LIN {X 0,Y 523.335,Z 480.946,A -85,B 0,C 180,E1 -4767.691,E2 -4767.691} C_VEL
LIN {X 0,Y 523.25,Z 482.542,A -85,B 0,C 180,E1 -4769.231,E2 -4769.231} C_VEL
LIN {X 0,Y 523.247,Z 482.758,A -85,B 0,C 180,E1 -4770,E2 -4770} C_VEL
LIN {X 0,Y 523.275,Z 481.937,A -85,B 0,C 180,E1 -4771.539,E2 -4771.539} C_VEL
LIN {X 0,Y 523.335,Z 480.945,A -85,B 0,C 180,E1 -4772.309,E2 -4772.309} C_VEL
LIN {X 0,Y 523.369,Z 479.554,A -85,B 0,C 180,E1 -4773.079,E2 -4773.079} C_VEL
LIN {X 0,Y 523.425,Z 476.628,A -85,B 0,C 180,E1 -4774.235,E2 -4774.235} C_VEL
LIN {X 0,Y 523.462,Z 472.665,A -85,B 0,C 180,E1 -4775.393,E2 -4775.393} C_VEL
LIN {X 0,Y 523.507,Z 466.591,A -85,B 0,C 180,E1 -4776.742,E2 -4776.742} C_VEL
LIN {X 0,Y 523.676,Z 459.903,A -85,B 0,C 180,E1 -4777.907,E2 -4777.907} C_VEL
LIN {X 0,Y 523.862,Z 451.631,A -85,B 0,C 180,E1 -4779.07,E2 -4779.07} C_VEL
LIN {X 0,Y 524.082,Z 443.149,A -85,B 0,C 180,E1 -4780.04,E2 -4780.04} C_VEL
LIN {X 0,Y 524.37,Z 432.664,A -85,B 0,C 180,E1 -4781.011,E2 -4781.011} C_VEL
LIN {X 0,Y 524.659,Z 422.41,A -85,B 0,C 180,E1 -4781.779,E2 -4781.779} C_VEL
LIN {X 0,Y 524.937,Z 410.907,A -85,B 0,C 180,E1 -4782.468,E2 -4782.468} C_VEL
LIN {X 0,Y 525.162,Z 399.206,A -85,B 0,C 180,E1 -4783.003,E2 -4783.003} C_VEL
LIN {X 0,Y 525.398,Z 385.719,A -85,B 0,C 180,E1 -4783.44,E2 -4783.44} C_VEL
LIN {X 0,Y 525.556,Z 372.288,A -85,B 0,C 180,E1 -4783.706,E2 -4783.706} C_VEL
LIN {X 0,Y 525.863,Z 280.733,A -85,B 0,C 180,E1 -4784.966,E2 -4784.966} C_VEL
LIN {X 0,Y 524.292,Z 270.902,A -85,B 0,C 180,E1 -4785.169,E2 -4785.169} C_VEL
LIN {X 0,Y 524.363,Z 264.633,A -85,B 0,C 180,E1 -4786.148,E2 -4786.148} C_VEL
LIN {X 0,Y 524.69,Z 248.812,A -85,B 0,C 180,E1 -4788.752,E2 -4788.752} C_VEL
LIN {X 0,Y 525.199,Z 230.548,A -85,B 0,C 180,E1 -4791.798,E2 -4791.798} C_VEL
LIN {X 0,Y 524.728,Z 225.858,A -85,B 0,C 180,E1 -4792.616,E2 -4792.616} C_VEL
LIN {X 0,Y 523.966,Z 221.81,A -85,B 0,C 180,E1 -4793.387,E2 -4793.387} C_VEL
LIN {X 0,Y 523.946,Z 221.721,A -85,B 0,C 180,E1 -4796.273,E2 -4796.273} C_VEL
LIN {X 0,Y 523.937,Z 221.717,A -85,B 0,C 180,E1 -4798.875,E2 -4798.875} C_VEL
LIN {X 0,Y 523.927,Z 221.72,A -85,B 0,C 180,E1 -4801.544,E2 -4801.544} C_VEL
LIN {X 0,Y 523.939,Z 221.722,A -85,B 0,C 180,E1 -4804.29,E2 -4804.29} C_VEL
LIN {X 0,Y 523.913,Z 221.719,A -85,B 0,C 180,E1 -4807.132,E2 -4807.132} C_VEL
LIN {X 0,Y 523.923,Z 221.723,A -85,B 0,C 180,E1 -4810.126,E2 -4810.126} C_VEL
LIN {X 0,Y 523.926,Z 221.721,A -85,B 0,C 180,E1 -4812.456,E2 -4812.456} C_VEL
LIN {X 0,Y 523.947,Z 221.715,A -85,B 0,C 180,E1 -4815.31,E2 -4815.31} C_VEL
LIN {X 0,Y 523.95,Z 221.721,A -85,B 0,C 180,E1 -4818.691,E2 -4818.691} C_VEL
LIN {X 0,Y 523.922,Z 221.717,A -85,B 0,C 180,E1 -4821.896,E2 -4821.896} C_VEL
LIN {X 0,Y 523.927,Z 221.725,A -85,B 0,C 180,E1 -4824.911,E2 -4824.911} C_VEL
LIN {X 0,Y 523.943,Z 221.713,A -85,B 0,C 180,E1 -4827.678,E2 -4827.678} C_VEL
LIN {X 0,Y 523.945,Z 221.72,A -85,B 0,C 180,E1 -4830.678,E2 -4830.678} C_VEL
LIN {X 0,Y 523.912,Z 221.72,A -85,B 0,C 180,E1 -4833.723,E2 -4833.723} C_VEL
LIN {X 0,Y 523.916,Z 221.716,A -85,B 0,C 180,E1 -4836.267,E2 -4836.267} C_VEL
LIN {X 0,Y 523.951,Z 221.716,A -85,B 0,C 180,E1 -4838.764,E2 -4838.764} C_VEL
LIN {X 0,Y 523.953,Z 221.718,A -85,B 0,C 180,E1 -4841.218,E2 -4841.218} C_VEL
LIN {X 0,Y 523.934,Z 221.72,A -85,B 0,C 180,E1 -4843.636,E2 -4843.636} C_VEL
LIN {X 0,Y 523.935,Z 221.719,A -85,B 0,C 180,E1 -4846.025,E2 -4846.025} C_VEL
LIN {X 0,Y 523.997,Z 221.709,A -85,B 0,C 180,E1 -4849.174,E2 -4849.174} C_VEL
LIN {X 0,Y 524.002,Z 221.709,A -85,B 0,C 180,E1 -4852.289,E2 -4852.289} C_VEL
LIN {X 0,Y 524.071,Z 221.698,A -85,B 0,C 180,E1 -4854.61,E2 -4854.61} C_VEL
LIN {X 0,Y 524.11,Z 221.699,A -85,B 0,C 180,E1 -4857.691,E2 -4857.691} C_VEL
LIN {X 0,Y 524.116,Z 221.694,A -85,B 0,C 180,E1 -4860.765,E2 -4860.765} C_VEL
LIN {X 0,Y 524.037,Z 221.7,A -85,B 0,C 180,E1 -4863.072,E2 -4863.072} C_VEL
LIN {X 0,Y 524.025,Z 221.713,A -85,B 0,C 180,E1 -4866.156,E2 -4866.156} C_VEL
LIN {X 0,Y 523.982,Z 221.71,A -85,B 0,C 180,E1 -4869.258,E2 -4869.258} C_VEL
LIN {X 0,Y 523.993,Z 221.706,A -85,B 0,C 180,E1 -4871.734,E2 -4871.734} C_VEL
LIN {X 0,Y 523.985,Z 221.711,A -85,B 0,C 180,E1 -4875.049,E2 -4875.049} C_VEL
LIN {X 0,Y 523.936,Z 221.716,A -85,B 0,C 180,E1 -4877.965,E2 -4877.965} C_VEL
LIN {X 0,Y 523.96,Z 221.717,A -85,B 0,C 180,E1 -4880.406,E2 -4880.406} C_VEL
LIN {X 0,Y 523.905,Z 221.728,A -85,B 0,C 180,E1 -4882.889,E2 -4882.889} C_VEL
LIN {X 0,Y 523.935,Z 221.713,A -85,B 0,C 180,E1 -4885.414,E2 -4885.414} C_VEL
LIN {X 0,Y 523.951,Z 221.714,A -85,B 0,C 180,E1 -4887.995,E2 -4887.995} C_VEL
LIN {X 0,Y 523.923,Z 221.721,A -85,B 0,C 180,E1 -4890.851,E2 -4890.851} C_VEL
LIN {X 0,Y 523.938,Z 221.718,A -85,B 0,C 180,E1 -4893.731,E2 -4893.731} C_VEL
LIN {X 0,Y 523.896,Z 221.721,A -85,B 0,C 180,E1 -4896.4,E2 -4896.4} C_VEL
LIN {X 0,Y 523.934,Z 221.719,A -85,B 0,C 180,E1 -4899.077,E2 -4899.077} C_VEL
LIN {X 0,Y 523.935,Z 221.719,A -85,B 0,C 180,E1 -4902.114,E2 -4902.114} C_VEL
LIN {X 0,Y 523.922,Z 221.723,A -85,B 0,C 180,E1 -4905.305,E2 -4905.305} C_VEL
LIN {X 0,Y 523.889,Z 221.724,A -85,B 0,C 180,E1 -4906.894,E2 -4906.894} C_VEL
LIN {X 0,Y 523.214,Z 221.816,A -85,B 0,C 180,E1 -4907.536,E2 -4907.536} C_VEL
LIN {X 0,Y 520.346,Z 222.167,A -85,B 0,C 180,E1 -4908.578,E2 -4908.578} C_VEL
LIN {X 0,Y 517.961,Z 222.468,A -85,B 0,C 180,E1 -4909.417,E2 -4909.417} C_VEL
LIN {X 0,Y 516.989,Z 222.591,A -85,B 0,C 180,E1 -4910.065,E2 -4910.065} C_VEL
LIN {X 0,Y 516.937,Z 222.597,A -85,B 0,C 180,E1 -4910.284,E2 -4910.284} C_VEL
LIN {X 0,Y 516.957,Z 222.758,A -85,B 0,C 180,E1 -4910.489,E2 -4910.489} C_VEL
LIN {X 0,Y 517.786,Z 229.073,A -85,B 0,C 180,E1 -4911.688,E2 -4911.688} C_VEL
LIN {X 0,Y 517.418,Z 247.056,A -85,B 0,C 180,E1 -4914.887,E2 -4914.887} C_VEL
LIN {X 0,Y 517.241,Z 257.287,A -85,B 0,C 180,E1 -4916.658,E2 -4916.658} C_VEL
LIN {X 0,Y 518.403,Z 263.881,A -85,B 0,C 180,E1 -4916.818,E2 -4916.818} C_VEL
LIN {X 0,Y 519.11,Z 269.37,A -85,B 0,C 180,E1 -4916.917,E2 -4916.917} C_VEL
LIN {X 0,Y 518.609,Z 364.635,A -85,B 0,C 180,E1 -4918.261,E2 -4918.261} C_VEL
LIN {X 0,Y 518.423,Z 378.207,A -85,B 0,C 180,E1 -4918.618,E2 -4918.618} C_VEL
LIN {X 0,Y 518.169,Z 390.312,A -85,B 0,C 180,E1 -4919.089,E2 -4919.089} C_VEL
LIN {X 0,Y 517.891,Z 402.731,A -85,B 0,C 180,E1 -4919.748,E2 -4919.748} C_VEL
LIN {X 0,Y 517.6,Z 413.253,A -85,B 0,C 180,E1 -4920.465,E2 -4920.465} C_VEL
LIN {X 0,Y 517.267,Z 424.093,A -85,B 0,C 180,E1 -4921.384,E2 -4921.384} C_VEL
LIN {X 0,Y 517.051,Z 432.491,A -85,B 0,C 180,E1 -4922.259,E2 -4922.259} C_VEL
LIN {X 0,Y 516.749,Z 440.994,A -85,B 0,C 180,E1 -4923.332,E2 -4923.332} C_VEL
LIN {X 0,Y 516.558,Z 449.157,A -85,B 0,C 180,E1 -4924.623,E2 -4924.623} C_VEL
LIN {X 0,Y 516.41,Z 455.564,A -85,B 0,C 180,E1 -4925.903,E2 -4925.903} C_VEL
LIN {X 0,Y 516.327,Z 460.463,A -85,B 0,C 180,E1 -4927.174,E2 -4927.174} C_VEL
LIN {X 0,Y 516.259,Z 464.071,A -85,B 0,C 180,E1 -4928.435,E2 -4928.435} C_VEL
LIN {X 0,Y 516.237,Z 466.879,A -85,B 0,C 180,E1 -4929.927,E2 -4929.927} C_VEL
LIN {X 0,Y 516.172,Z 467.939,A -85,B 0,C 180,E1 -4930.927,E2 -4930.927} C_VEL
LIN {X 0,Y 516.18,Z 468.302,A -85,B 0,C 180,E1 -4932.359,E2 -4932.359} C_VEL
LIN {X 0,Y 516.19,Z 467.766,A -85,B 0,C 180,E1 -4933.386,E2 -4933.386} C_VEL
LIN {X 0,Y 516.209,Z 466.822,A -85,B 0,C 180,E1 -4934.199,E2 -4934.199} C_VEL
LIN {X 0,Y 516.252,Z 465.267,A -85,B 0,C 180,E1 -4935.117,E2 -4935.117} C_VEL
LIN {X 0,Y 516.304,Z 462.587,A -85,B 0,C 180,E1 -4936.219,E2 -4936.219} C_VEL
LIN {X 0,Y 516.341,Z 458.654,A -85,B 0,C 180,E1 -4937.421,E2 -4937.421} C_VEL
LIN {X 0,Y 516.533,Z 453.072,A -85,B 0,C 180,E1 -4938.722,E2 -4938.722} C_VEL
LIN {X 0,Y 516.64,Z 445.925,A -85,B 0,C 180,E1 -4940.012,E2 -4940.012} C_VEL
LIN {X 0,Y 516.839,Z 437.679,A -85,B 0,C 180,E1 -4941.2,E2 -4941.2} C_VEL
LIN {X 0,Y 517.127,Z 429.239,A -85,B 0,C 180,E1 -4942.189,E2 -4942.189} C_VEL
LIN {X 0,Y 517.396,Z 418.866,A -85,B 0,C 180,E1 -4943.174,E2 -4943.174} C_VEL
LIN {X 0,Y 517.748,Z 407.176,A -85,B 0,C 180,E1 -4944.059,E2 -4944.059} C_VEL
LIN {X 0,Y 518.06,Z 395.541,A -85,B 0,C 180,E1 -4944.746,E2 -4944.746} C_VEL
LIN {X 0,Y 518.319,Z 383.483,A -85,B 0,C 180,E1 -4945.285,E2 -4945.285} C_VEL
LIN {X 0,Y 518.506,Z 370.393,A -85,B 0,C 180,E1 -4945.7,E2 -4945.7} C_VEL
LIN {X 0,Y 518.683,Z 357.572,A -85,B 0,C 180,E1 -4945.945,E2 -4945.945} C_VEL
LIN {X 0,Y 519.048,Z 267.685,A -85,B 0,C 180,E1 -4947.199,E2 -4947.199} C_VEL
LIN {X 0,Y 517.307,Z 257.515,A -85,B 0,C 180,E1 -4947.42,E2 -4947.42} C_VEL
LIN {X 0,Y 517.358,Z 249.489,A -85,B 0,C 180,E1 -4948.832,E2 -4948.832} C_VEL
LIN {X 0,Y 517.835,Z 233.569,A -85,B 0,C 180,E1 -4951.75,E2 -4951.75} C_VEL
LIN {X 0,Y 517.797,Z 227.316,A -85,B 0,C 180,E1 -4952.917,E2 -4952.917} C_VEL
LIN {X 0,Y 516.879,Z 222.661,A -85,B 0,C 180,E1 -4953.874,E2 -4953.874} C_VEL
LIN {X 0,Y 517.008,Z 222.587,A -85,B 0,C 180,E1 -4956.243,E2 -4956.243} C_VEL
LIN {X 0,Y 516.947,Z 222.595,A -85,B 0,C 180,E1 -4958.6,E2 -4958.6} C_VEL
LIN {X 0,Y 516.967,Z 222.585,A -85,B 0,C 180,E1 -4961.844,E2 -4961.844} C_VEL
LIN {X 0,Y 516.928,Z 222.592,A -85,B 0,C 180,E1 -4965.162,E2 -4965.162} C_VEL
LIN {X 0,Y 516.883,Z 222.594,A -85,B 0,C 180,E1 -4968.223,E2 -4968.223} C_VEL
LIN {X 0,Y 516.888,Z 222.595,A -85,B 0,C 180,E1 -4970.702,E2 -4970.702} C_VEL
LIN {X 0,Y 516.873,Z 222.601,A -85,B 0,C 180,E1 -4973.223,E2 -4973.223} C_VEL
LIN {X 0,Y 516.909,Z 222.582,A -85,B 0,C 180,E1 -4976.202,E2 -4976.202} C_VEL
LIN {X 0,Y 516.9,Z 222.596,A -85,B 0,C 180,E1 -4979.305,E2 -4979.305} C_VEL
LIN {X 0,Y 516.86,Z 222.599,A -85,B 0,C 180,E1 -4982.025,E2 -4982.025} C_VEL
LIN {X 0,Y 516.894,Z 222.591,A -85,B 0,C 180,E1 -4984.823,E2 -4984.823} C_VEL
LIN {X 0,Y 516.857,Z 222.602,A -85,B 0,C 180,E1 -4987.949,E2 -4987.949} C_VEL
LIN {X 0,Y 516.885,Z 222.592,A -85,B 0,C 180,E1 -4990.741,E2 -4990.741} C_VEL
LIN {X 0,Y 516.918,Z 222.596,A -85,B 0,C 180,E1 -4993.905,E2 -4993.905} C_VEL
LIN {X 0,Y 516.92,Z 222.597,A -85,B 0,C 180,E1 -4996.108,E2 -4996.108} C_VEL
LIN {X 0,Y 516.884,Z 222.592,A -85,B 0,C 180,E1 -4999.265,E2 -4999.265} C_VEL
LIN {X 0,Y 516.858,Z 222.596,A -85,B 0,C 180,E1 -5002.059,E2 -5002.059} C_VEL
LIN {X 0,Y 516.876,Z 222.594,A -85,B 0,C 180,E1 -5005.181,E2 -5005.181} C_VEL
LIN {X 0,Y 516.859,Z 222.6,A -85,B 0,C 180,E1 -5007.98,E2 -5007.98} C_VEL
LIN {X 0,Y 516.913,Z 222.588,A -85,B 0,C 180,E1 -5010.7,E2 -5010.7} C_VEL
LIN {X 0,Y 516.924,Z 222.582,A -85,B 0,C 180,E1 -5013.807,E2 -5013.807} C_VEL
LIN {X 0,Y 516.874,Z 222.604,A -85,B 0,C 180,E1 -5016.782,E2 -5016.782} C_VEL
LIN {X 0,Y 516.923,Z 222.588,A -85,B 0,C 180,E1 -5019.735,E2 -5019.735} C_VEL
LIN {X 0,Y 516.917,Z 222.589,A -85,B 0,C 180,E1 -5022.6,E2 -5022.6} C_VEL
LIN {X 0,Y 516.929,Z 222.585,A -85,B 0,C 180,E1 -5025.034,E2 -5025.034} C_VEL
LIN {X 0,Y 516.994,Z 222.577,A -85,B 0,C 180,E1 -5028.238,E2 -5028.238} C_VEL
LIN {X 0,Y 516.965,Z 222.592,A -85,B 0,C 180,E1 -5031.404,E2 -5031.404} C_VEL
LIN {X 0,Y 517.008,Z 222.58,A -85,B 0,C 180,E1 -5033.761,E2 -5033.761} C_VEL
LIN {X 0,Y 517.079,Z 222.566,A -85,B 0,C 180,E1 -5037.667,E2 -5037.667} C_VEL
LIN {X 0,Y 517.09,Z 222.564,A -85,B 0,C 180,E1 -5040.782,E2 -5040.782} C_VEL
LIN {X 0,Y 517.01,Z 222.578,A -85,B 0,C 180,E1 -5043.12,E2 -5043.12} C_VEL
LIN {X 0,Y 516.992,Z 222.583,A -85,B 0,C 180,E1 -5046.247,E2 -5046.247} C_VEL
LIN {X 0,Y 516.965,Z 222.578,A -85,B 0,C 180,E1 -5048.604,E2 -5048.604} C_VEL
LIN {X 0,Y 516.954,Z 222.582,A -85,B 0,C 180,E1 -5051.81,E2 -5051.81} C_VEL
LIN {X 0,Y 516.948,Z 222.586,A -85,B 0,C 180,E1 -5055.149,E2 -5055.149} C_VEL
LIN {X 0,Y 516.92,Z 222.596,A -85,B 0,C 180,E1 -5058.225,E2 -5058.225} C_VEL
LIN {X 0,Y 516.917,Z 222.59,A -85,B 0,C 180,E1 -5060.704,E2 -5060.704} C_VEL
LIN {X 0,Y 516.906,Z 222.592,A -85,B 0,C 180,E1 -5064.075,E2 -5064.075} C_VEL
LIN {X 0,Y 516.909,Z 222.6,A -85,B 0,C 180,E1 -5066.661,E2 -5066.661} C_VEL
LIN {X 0,Y 516.915,Z 222.585,A -85,B 0,C 180,E1 -5069.525,E2 -5069.525} C_VEL
LIN {X 0,Y 516.9,Z 222.595,A -85,B 0,C 180,E1 -5072.545,E2 -5072.545} C_VEL
LIN {X 0,Y 516.869,Z 222.6,A -85,B 0,C 180,E1 -5075.331,E2 -5075.331} C_VEL
LIN {X 0,Y 516.884,Z 222.592,A -85,B 0,C 180,E1 -5077.944,E2 -5077.944} C_VEL
LIN {X 0,Y 516.889,Z 222.596,A -85,B 0,C 180,E1 -5080.743,E2 -5080.743} C_VEL
LIN {X 0,Y 516.888,Z 222.586,A -85,B 0,C 180,E1 -5083.905,E2 -5083.905} C_VEL
LIN {X 0,Y 516.887,Z 222.589,A -85,B 0,C 180,E1 -5086.109,E2 -5086.109} C_VEL
LIN {X 0,Y 516.889,Z 222.597,A -85,B 0,C 180,E1 -5089.259,E2 -5089.259} C_VEL
LIN {X 0,Y 516.867,Z 222.597,A -85,B 0,C 180,E1 -5092.275,E2 -5092.275} C_VEL
LIN {X 0,Y 516.888,Z 222.595,A -85,B 0,C 180,E1 -5095.176,E2 -5095.176} C_VEL
LIN {X 0,Y 516.88,Z 222.603,A -85,B 0,C 180,E1 -5097.976,E2 -5097.976} C_VEL
LIN {X 0,Y 516.926,Z 222.592,A -85,B 0,C 180,E1 -5100.696,E2 -5100.696} C_VEL
LIN {X 0,Y 516.913,Z 222.594,A -85,B 0,C 180,E1 -5103.342,E2 -5103.342} C_VEL
LIN {X 0,Y 516.939,Z 222.71,A -85,B 0,C 180,E1 -5106.409,E2 -5106.409} C_VEL
LIN {X 0,Y 518.257,Z 230.708,A -85,B 0,C 180,E1 -5107.895,E2 -5107.895} C_VEL
LIN {X 0,Y 517.79,Z 248.894,A -85,B 0,C 180,E1 -5110.989,E2 -5110.989} C_VEL
LIN {X 0,Y 517.375,Z 265.834,A -85,B 0,C 180,E1 -5113.831,E2 -5113.831} C_VEL
LIN {X 0,Y 517.277,Z 270.785,A -85,B 0,C 180,E1 -5114.615,E2 -5114.615} C_VEL
LIN {X 0,Y 518.992,Z 281.529,A -85,B 0,C 180,E1 -5114.844,E2 -5114.844} C_VEL
LIN {X 0,Y 518.631,Z 378.172,A -85,B 0,C 180,E1 -5116.207,E2 -5116.207} C_VEL
LIN {X 0,Y 518.407,Z 391.541,A -85,B 0,C 180,E1 -5116.551,E2 -5116.551} C_VEL
LIN {X 0,Y 518.138,Z 404.876,A -85,B 0,C 180,E1 -5117.068,E2 -5117.068} C_VEL
LIN {X 0,Y 517.878,Z 416.116,A -85,B 0,C 180,E1 -5117.662,E2 -5117.662} C_VEL
LIN {X 0,Y 517.568,Z 427.664,A -85,B 0,C 180,E1 -5118.446,E2 -5118.446} C_VEL
LIN {X 0,Y 517.205,Z 438.107,A -85,B 0,C 180,E1 -5119.331,E2 -5119.331} C_VEL
LIN {X 0,Y 516.98,Z 446.645,A -85,B 0,C 180,E1 -5120.217,E2 -5120.217} C_VEL
LIN {X 0,Y 516.755,Z 454.519,A -85,B 0,C 180,E1 -5121.199,E2 -5121.199} C_VEL
LIN {X 0,Y 516.552,Z 462.207,A -85,B 0,C 180,E1 -5122.377,E2 -5122.377} C_VEL
LIN {X 0,Y 516.405,Z 469.291,A -85,B 0,C 180,E1 -5123.75,E2 -5123.75} C_VEL
LIN {X 0,Y 516.314,Z 474.002,A -85,B 0,C 180,E1 -5124.924,E2 -5124.924} C_VEL
LIN {X 0,Y 516.353,Z 477.601,A -85,B 0,C 180,E1 -5126.098,E2 -5126.098} C_VEL
LIN {X 0,Y 516.284,Z 479.456,A -85,B 0,C 180,E1 -5126.879,E2 -5126.879} C_VEL
LIN {X 0,Y 516.262,Z 480.847,A -85,B 0,C 180,E1 -5127.66,E2 -5127.66} C_VEL
LIN {X 0,Y 516.161,Z 482.444,A -85,B 0,C 180,E1 -5129.22,E2 -5129.22} C_VEL
LIN {X 0,Y 516.155,Z 482.66,A -85,B 0,C 180,E1 -5130,E2 -5130} C_VEL
LIN {X 0,Y 516.193,Z 481.838,A -85,B 0,C 180,E1 -5131.561,E2 -5131.561} C_VEL
LIN {X 0,Y 516.262,Z 480.846,A -85,B 0,C 180,E1 -5132.341,E2 -5132.341} C_VEL
LIN {X 0,Y 516.284,Z 479.454,A -85,B 0,C 180,E1 -5133.122,E2 -5133.122} C_VEL
LIN {X 0,Y 516.314,Z 476.526,A -85,B 0,C 180,E1 -5134.294,E2 -5134.294} C_VEL
LIN {X 0,Y 516.399,Z 472.562,A -85,B 0,C 180,E1 -5135.467,E2 -5135.467} C_VEL
LIN {X 0,Y 516.426,Z 467.354,A -85,B 0,C 180,E1 -5136.665,E2 -5136.665} C_VEL
LIN {X 0,Y 516.585,Z 461.031,A -85,B 0,C 180,E1 -5137.819,E2 -5137.819} C_VEL
LIN {X 0,Y 516.773,Z 453.011,A -85,B 0,C 180,E1 -5138.998,E2 -5138.998} C_VEL
LIN {X 0,Y 517.027,Z 444.837,A -85,B 0,C 180,E1 -5139.981,E2 -5139.981} C_VEL
LIN {X 0,Y 517.337,Z 434.865,A -85,B 0,C 180,E1 -5140.964,E2 -5140.964} C_VEL
LIN {X 0,Y 517.649,Z 425.021,A -85,B 0,C 180,E1 -5141.751,E2 -5141.751} C_VEL
LIN {X 0,Y 517.917,Z 413.872,A -85,B 0,C 180,E1 -5142.466,E2 -5142.466} C_VEL
LIN {X 0,Y 518.192,Z 401.434,A -85,B 0,C 180,E1 -5143.081,E2 -5143.081} C_VEL
LIN {X 0,Y 518.487,Z 388.315,A -85,B 0,C 180,E1 -5143.547,E2 -5143.547} C_VEL
LIN {X 0,Y 518.654,Z 375.175,A -85,B 0,C 180,E1 -5143.842,E2 -5143.842} C_VEL
LIN {X 0,Y 518.988,Z 281.442,A -85,B 0,C 180,E1 -5145.157,E2 -5145.157} C_VEL
LIN {X 0,Y 517.261,Z 270.8,A -85,B 0,C 180,E1 -5145.38,E2 -5145.38} C_VEL
LIN {X 0,Y 517.493,Z 259.66,A -85,B 0,C 180,E1 -5147.181,E2 -5147.181} C_VEL
LIN {X 0,Y 517.948,Z 241.633,A -85,B 0,C 180,E1 -5150.206,E2 -5150.206} C_VEL
LIN {X 0,Y 518.247,Z 230.459,A -85,B 0,C 180,E1 -5152.106,E2 -5152.106} C_VEL
LIN {X 0,Y 516.934,Z 222.727,A -85,B 0,C 180,E1 -5153.539,E2 -5153.539} C_VEL
LIN {X 0,Y 516.914,Z 222.594,A -85,B 0,C 180,E1 -5156.659,E2 -5156.659} C_VEL
LIN {X 0,Y 516.916,Z 222.595,A -85,B 0,C 180,E1 -5159.522,E2 -5159.522} C_VEL
LIN {X 0,Y 516.905,Z 222.593,A -85,B 0,C 180,E1 -5162.542,E2 -5162.542} C_VEL
LIN {X 0,Y 516.871,Z 222.596,A -85,B 0,C 180,E1 -5165.328,E2 -5165.328} C_VEL
LIN {X 0,Y 516.887,Z 222.601,A -85,B 0,C 180,E1 -5167.942,E2 -5167.942} C_VEL
LIN {X 0,Y 516.874,Z 222.599,A -85,B 0,C 180,E1 -5170.743,E2 -5170.743} C_VEL
LIN {X 0,Y 516.864,Z 222.598,A -85,B 0,C 180,E1 -5172.833,E2 -5172.833} C_VEL
LIN {X 0,Y 516.906,Z 222.594,A -85,B 0,C 180,E1 -5175.006,E2 -5175.006} C_VEL
LIN {X 0,Y 516.913,Z 222.592,A -85,B 0,C 180,E1 -5178.399,E2 -5178.399} C_VEL
LIN {X 0,Y 516.888,Z 222.594,A -85,B 0,C 180,E1 -5181.282,E2 -5181.282} C_VEL
LIN {X 0,Y 516.875,Z 222.597,A -85,B 0,C 180,E1 -5184.218,E2 -5184.218} C_VEL
LIN {X 0,Y 516.89,Z 222.599,A -85,B 0,C 180,E1 -5187.05,E2 -5187.05} C_VEL
LIN {X 0,Y 516.876,Z 222.596,A -85,B 0,C 180,E1 -5189.793,E2 -5189.793} C_VEL
LIN {X 0,Y 516.884,Z 222.594,A -85,B 0,C 180,E1 -5192.462,E2 -5192.462} C_VEL
LIN {X 0,Y 516.854,Z 222.606,A -85,B 0,C 180,E1 -5195.066,E2 -5195.066} C_VEL
LIN {X 0,Y 516.878,Z 222.599,A -85,B 0,C 180,E1 -5197.619,E2 -5197.619} C_VEL
LIN {X 0,Y 516.939,Z 222.585,A -85,B 0,C 180,E1 -5200.127,E2 -5200.127} C_VEL
LIN {X 0,Y 516.913,Z 222.591,A -85,B 0,C 180,E1 -5202.593,E2 -5202.593} C_VEL
LIN {X 0,Y 516.948,Z 222.585,A -85,B 0,C 180,E1 -5205.027,E2 -5205.027} C_VEL
LIN {X 0,Y 516.972,Z 222.582,A -85,B 0,C 180,E1 -5208.231,E2 -5208.231} C_VEL
LIN {X 0,Y 516.934,Z 222.592,A -85,B 0,C 180,E1 -5211.396,E2 -5211.396} C_VEL
LIN {X 0,Y 516.989,Z 222.587,A -85,B 0,C 180,E1 -5213.753,E2 -5213.753} C_VEL
LIN {X 0,Y 516.975,Z 222.582,A -85,B 0,C 180,E1 -5216.879,E2 -5216.879} C_VEL
LIN {X 0,Y 517.091,Z 222.566,A -85,B 0,C 180,E1 -5219.218,E2 -5219.218} C_VEL
LIN {X 0,Y 517.079,Z 222.573,A -85,B 0,C 180,E1 -5222.333,E2 -5222.333} C_VEL
LIN {X 0,Y 517.018,Z 222.578,A -85,B 0,C 180,E1 -5225.456,E2 -5225.456} C_VEL
LIN {X 0,Y 516.959,Z 222.591,A -85,B 0,C 180,E1 -5228.597,E2 -5228.597} C_VEL
LIN {X 0,Y 516.945,Z 222.585,A -85,B 0,C 180,E1 -5231.803,E2 -5231.803} C_VEL
LIN {X 0,Y 516.938,Z 222.588,A -85,B 0,C 180,E1 -5235.143,E2 -5235.143} C_VEL
LIN {X 0,Y 516.905,Z 222.594,A -85,B 0,C 180,E1 -5238.218,E2 -5238.218} C_VEL
LIN {X 0,Y 516.901,Z 222.601,A -85,B 0,C 180,E1 -5240.697,E2 -5240.697} C_VEL
LIN {X 0,Y 516.859,Z 222.602,A -85,B 0,C 180,E1 -5243.219,E2 -5243.219} C_VEL
LIN {X 0,Y 516.925,Z 222.584,A -85,B 0,C 180,E1 -5246.192,E2 -5246.192} C_VEL
LIN {X 0,Y 516.901,Z 222.597,A -85,B 0,C 180,E1 -5249.3,E2 -5249.3} C_VEL
LIN {X 0,Y 516.875,Z 222.596,A -85,B 0,C 180,E1 -5252.54,E2 -5252.54} C_VEL
LIN {X 0,Y 516.857,Z 222.603,A -85,B 0,C 180,E1 -5255.328,E2 -5255.328} C_VEL
LIN {X 0,Y 516.858,Z 222.598,A -85,B 0,C 180,E1 -5257.94,E2 -5257.94} C_VEL
LIN {X 0,Y 516.888,Z 222.595,A -85,B 0,C 180,E1 -5260.734,E2 -5260.734} C_VEL
LIN {X 0,Y 516.85,Z 222.605,A -85,B 0,C 180,E1 -5263.899,E2 -5263.899} C_VEL
LIN {X 0,Y 516.848,Z 222.604,A -85,B 0,C 180,E1 -5266.103,E2 -5266.103} C_VEL
LIN {X 0,Y 516.884,Z 222.6,A -85,B 0,C 180,E1 -5269.258,E2 -5269.258} C_VEL
LIN {X 0,Y 516.937,Z 222.597,A -85,B 0,C 180,E1 -5270.284,E2 -5270.284} C_VEL
LIN {X 0,Y 516.819,Z 223.447,A -85,B 0,C 180,E1 -5270.614,E2 -5270.614} C_VEL
LIN {X 0,Y 516.039,Z 226.233,A -85,B 0,C 180,E1 -5271.103,E2 -5271.103} C_VEL
LIN {X 0,Y 511.302,Z 236.065,A -85,B 0,C 180,E1 -5272.666,E2 -5272.666} C_VEL
LIN {X 0,Y 510.587,Z 239.154,A -85,B 0,C 180,E1 -5273.217,E2 -5273.217} C_VEL
LIN {X 0,Y 510.32,Z 254.146,A -85,B 0,C 180,E1 -5275.906,E2 -5275.906} C_VEL
LIN {X 0,Y 510.255,Z 257.328,A -85,B 0,C 180,E1 -5276.435,E2 -5276.435} C_VEL
LIN {X 0,Y 511.252,Z 263.108,A -85,B 0,C 180,E1 -5276.587,E2 -5276.587} C_VEL
LIN {X 0,Y 512.281,Z 269.989,A -85,B 0,C 180,E1 -5276.718,E2 -5276.718} C_VEL
LIN {X 0,Y 511.718,Z 365.353,A -85,B 0,C 180,E1 -5278.087,E2 -5278.087} C_VEL
LIN {X 0,Y 511.509,Z 379.166,A -85,B 0,C 180,E1 -5278.463,E2 -5278.463} C_VEL
LIN {X 0,Y 511.238,Z 391.625,A -85,B 0,C 180,E1 -5278.968,E2 -5278.968} C_VEL
LIN {X 0,Y 510.927,Z 403.195,A -85,B 0,C 180,E1 -5279.602,E2 -5279.602} C_VEL
LIN {X 0,Y 510.584,Z 414.686,A -85,B 0,C 180,E1 -5280.409,E2 -5280.409} C_VEL
LIN {X 0,Y 510.219,Z 425.514,A -85,B 0,C 180,E1 -5281.366,E2 -5281.366} C_VEL
LIN {X 0,Y 509.99,Z 433.94,A -85,B 0,C 180,E1 -5282.283,E2 -5282.283} C_VEL
LIN {X 0,Y 509.681,Z 441.999,A -85,B 0,C 180,E1 -5283.345,E2 -5283.345} C_VEL
LIN {X 0,Y 509.483,Z 450.166,A -85,B 0,C 180,E1 -5284.683,E2 -5284.683} C_VEL
LIN {X 0,Y 509.334,Z 456.399,A -85,B 0,C 180,E1 -5285.995,E2 -5285.995} C_VEL
LIN {X 0,Y 509.229,Z 461.063,A -85,B 0,C 180,E1 -5287.267,E2 -5287.267} C_VEL
LIN {X 0,Y 509.182,Z 463.515,A -85,B 0,C 180,E1 -5288.12,E2 -5288.12} C_VEL
LIN {X 0,Y 509.143,Z 465.442,A -85,B 0,C 180,E1 -5288.968,E2 -5288.968} C_VEL
LIN {X 0,Y 509.147,Z 466.858,A -85,B 0,C 180,E1 -5289.813,E2 -5289.813} C_VEL
LIN {X 0,Y 509.109,Z 467.834,A -85,B 0,C 180,E1 -5290.652,E2 -5290.652} C_VEL
LIN {X 0,Y 509.072,Z 468.353,A -85,B 0,C 180,E1 -5291.486,E2 -5291.486} C_VEL
LIN {X 0,Y 509.102,Z 468.409,A -85,B 0,C 180,E1 -5292.32,E2 -5292.32} C_VEL
LIN {X 0,Y 509.091,Z 468.053,A -85,B 0,C 180,E1 -5293.148,E2 -5293.148} C_VEL
LIN {X 0,Y 509.096,Z 467.28,A -85,B 0,C 180,E1 -5293.972,E2 -5293.972} C_VEL
LIN {X 0,Y 509.18,Z 465.595,A -85,B 0,C 180,E1 -5295.033,E2 -5295.033} C_VEL
LIN {X 0,Y 509.202,Z 462.271,A -85,B 0,C 180,E1 -5296.43,E2 -5296.43} C_VEL
LIN {X 0,Y 509.288,Z 458.192,A -85,B 0,C 180,E1 -5297.649,E2 -5297.649} C_VEL
LIN {X 0,Y 509.443,Z 451.908,A -85,B 0,C 180,E1 -5299.065,E2 -5299.065} C_VEL
LIN {X 0,Y 509.613,Z 445.083,A -85,B 0,C 180,E1 -5300.274,E2 -5300.274} C_VEL
LIN {X 0,Y 509.924,Z 436.587,A -85,B 0,C 180,E1 -5301.479,E2 -5301.479} C_VEL
LIN {X 0,Y 510.185,Z 426.496,A -85,B 0,C 180,E1 -5302.622,E2 -5302.622} C_VEL
LIN {X 0,Y 510.546,Z 415.986,A -85,B 0,C 180,E1 -5303.578,E2 -5303.578} C_VEL
LIN {X 0,Y 510.881,Z 404.956,A -85,B 0,C 180,E1 -5304.375,E2 -5304.375} C_VEL
LIN {X 0,Y 511.235,Z 392.614,A -85,B 0,C 180,E1 -5305.071,E2 -5305.071} C_VEL
LIN {X 0,Y 511.483,Z 380.921,A -85,B 0,C 180,E1 -5305.567,E2 -5305.567} C_VEL
LIN {X 0,Y 511.675,Z 368.29,A -85,B 0,C 180,E1 -5305.939,E2 -5305.939} C_VEL
LIN {X 0,Y 511.802,Z 350.571,A -85,B 0,C 180,E1 -5306.235,E2 -5306.235} C_VEL
LIN {X 0,Y 512.128,Z 267.888,A -85,B 0,C 180,E1 -5307.407,E2 -5307.407} C_VEL
LIN {X 0,Y 510.317,Z 257.676,A -85,B 0,C 180,E1 -5307.632,E2 -5307.632} C_VEL
LIN {X 0,Y 510.307,Z 254.132,A -85,B 0,C 180,E1 -5308.224,E2 -5308.224} C_VEL
LIN {X 0,Y 510.721,Z 238.142,A -85,B 0,C 180,E1 -5311.182,E2 -5311.182} C_VEL
LIN {X 0,Y 511.007,Z 229.708,A -85,B 0,C 180,E1 -5312.759,E2 -5312.759} C_VEL
LIN {X 0,Y 509.83,Z 223.535,A -85,B 0,C 180,E1 -5314.026,E2 -5314.026} C_VEL
LIN {X 0,Y 509.973,Z 223.464,A -85,B 0,C 180,E1 -5316.329,E2 -5316.329} C_VEL
LIN {X 0,Y 509.919,Z 223.469,A -85,B 0,C 180,E1 -5318.72,E2 -5318.72} C_VEL
LIN {X 0,Y 509.912,Z 223.465,A -85,B 0,C 180,E1 -5321.931,E2 -5321.931} C_VEL
LIN {X 0,Y 509.893,Z 223.467,A -85,B 0,C 180,E1 -5325.264,E2 -5325.264} C_VEL
LIN {X 0,Y 509.862,Z 223.467,A -85,B 0,C 180,E1 -5328.011,E2 -5328.011} C_VEL
LIN {X 0,Y 509.841,Z 223.478,A -85,B 0,C 180,E1 -5331.002,E2 -5331.002} C_VEL
LIN {X 0,Y 509.827,Z 223.474,A -85,B 0,C 180,E1 -5333.563,E2 -5333.563} C_VEL
LIN {X 0,Y 509.877,Z 223.458,A -85,B 0,C 180,E1 -5336.384,E2 -5336.384} C_VEL
LIN {X 0,Y 509.847,Z 223.467,A -85,B 0,C 180,E1 -5338.846,E2 -5338.846} C_VEL
LIN {X 0,Y 509.815,Z 223.482,A -85,B 0,C 180,E1 -5341.59,E2 -5341.59} C_VEL
LIN {X 0,Y 509.841,Z 223.469,A -85,B 0,C 180,E1 -5344.414,E2 -5344.414} C_VEL
LIN {X 0,Y 509.793,Z 223.481,A -85,B 0,C 180,E1 -5347.342,E2 -5347.342} C_VEL
LIN {X 0,Y 509.851,Z 223.469,A -85,B 0,C 180,E1 -5350.38,E2 -5350.38} C_VEL
LIN {X 0,Y 509.857,Z 223.469,A -85,B 0,C 180,E1 -5353.567,E2 -5353.567} C_VEL
LIN {X 0,Y 509.859,Z 223.472,A -85,B 0,C 180,E1 -5356.44,E2 -5356.44} C_VEL
LIN {X 0,Y 509.847,Z 223.471,A -85,B 0,C 180,E1 -5359.626,E2 -5359.626} C_VEL
LIN {X 0,Y 509.796,Z 223.475,A -85,B 0,C 180,E1 -5362.664,E2 -5362.664} C_VEL
LIN {X 0,Y 509.838,Z 223.473,A -85,B 0,C 180,E1 -5365.8,E2 -5365.8} C_VEL
LIN {X 0,Y 509.824,Z 223.475,A -85,B 0,C 180,E1 -5368.723,E2 -5368.723} C_VEL
LIN {X 0,Y 509.863,Z 223.46,A -85,B 0,C 180,E1 -5371.16,E2 -5371.16} C_VEL
LIN {X 0,Y 509.89,Z 223.458,A -85,B 0,C 180,E1 -5373.833,E2 -5373.833} C_VEL
LIN {X 0,Y 509.832,Z 223.475,A -85,B 0,C 180,E1 -5376.442,E2 -5376.442} C_VEL
LIN {X 0,Y 509.901,Z 223.463,A -85,B 0,C 180,E1 -5379.849,E2 -5379.849} C_VEL
LIN {X 0,Y 509.874,Z 223.463,A -85,B 0,C 180,E1 -5383.179,E2 -5383.179} C_VEL
LIN {X 0,Y 509.852,Z 223.463,A -85,B 0,C 180,E1 -5385.638,E2 -5385.638} C_VEL
LIN {X 0,Y 509.916,Z 223.463,A -85,B 0,C 180,E1 -5388.879,E2 -5388.879} C_VEL
LIN {X 0,Y 509.945,Z 223.458,A -85,B 0,C 180,E1 -5392.082,E2 -5392.082} C_VEL
LIN {X 0,Y 509.979,Z 223.45,A -85,B 0,C 180,E1 -5394.468,E2 -5394.468} C_VEL
LIN {X 0,Y 510.05,Z 223.441,A -85,B 0,C 180,E1 -5397.635,E2 -5397.635} C_VEL
LIN {X 0,Y 510.06,Z 223.44,A -85,B 0,C 180,E1 -5400.793,E2 -5400.793} C_VEL
LIN {X 0,Y 509.952,Z 223.458,A -85,B 0,C 180,E1 -5403.164,E2 -5403.164} C_VEL
LIN {X 0,Y 509.939,Z 223.46,A -85,B 0,C 180,E1 -5406.333,E2 -5406.333} C_VEL
LIN {X 0,Y 509.911,Z 223.455,A -85,B 0,C 180,E1 -5408.723,E2 -5408.723} C_VEL
LIN {X 0,Y 509.906,Z 223.461,A -85,B 0,C 180,E1 -5411.935,E2 -5411.935} C_VEL
LIN {X 0,Y 509.897,Z 223.464,A -85,B 0,C 180,E1 -5415.245,E2 -5415.245} C_VEL
LIN {X 0,Y 509.871,Z 223.47,A -85,B 0,C 180,E1 -5417.996,E2 -5417.996} C_VEL
LIN {X 0,Y 509.891,Z 223.466,A -85,B 0,C 180,E1 -5420.404,E2 -5420.404} C_VEL
LIN {X 0,Y 509.833,Z 223.471,A -85,B 0,C 180,E1 -5423.566,E2 -5423.566} C_VEL
LIN {X 0,Y 509.886,Z 223.471,A -85,B 0,C 180,E1 -5426.374,E2 -5426.374} C_VEL
LIN {X 0,Y 509.878,Z 223.47,A -85,B 0,C 180,E1 -5428.847,E2 -5428.847} C_VEL
LIN {X 0,Y 509.824,Z 223.474,A -85,B 0,C 180,E1 -5431.592,E2 -5431.592} C_VEL
LIN {X 0,Y 509.843,Z 223.473,A -85,B 0,C 180,E1 -5434.417,E2 -5434.417} C_VEL
LIN {X 0,Y 509.814,Z 223.48,A -85,B 0,C 180,E1 -5437.343,E2 -5437.343} C_VEL
LIN {X 0,Y 509.845,Z 223.471,A -85,B 0,C 180,E1 -5440.384,E2 -5440.384} C_VEL
LIN {X 0,Y 509.812,Z 223.477,A -85,B 0,C 180,E1 -5443.061,E2 -5443.061} C_VEL
LIN {X 0,Y 509.829,Z 223.471,A -85,B 0,C 180,E1 -5445.795,E2 -5445.795} C_VEL
LIN {X 0,Y 509.859,Z 223.469,A -85,B 0,C 180,E1 -5448.575,E2 -5448.575} C_VEL
LIN {X 0,Y 509.856,Z 223.474,A -85,B 0,C 180,E1 -5451.788,E2 -5451.788} C_VEL
LIN {X 0,Y 509.834,Z 223.473,A -85,B 0,C 180,E1 -5454.623,E2 -5454.623} C_VEL
LIN {X 0,Y 509.868,Z 223.472,A -85,B 0,C 180,E1 -5457.482,E2 -5457.482} C_VEL
LIN {X 0,Y 509.865,Z 223.475,A -85,B 0,C 180,E1 -5460.275,E2 -5460.275} C_VEL
LIN {X 0,Y 509.88,Z 223.47,A -85,B 0,C 180,E1 -5462.945,E2 -5462.945} C_VEL
LIN {X 0,Y 509.868,Z 223.558,A -85,B 0,C 180,E1 -5466.223,E2 -5466.223} C_VEL
LIN {X 0,Y 511.163,Z 230.597,A -85,B 0,C 180,E1 -5467.572,E2 -5467.572} C_VEL
LIN {X 0,Y 511.1,Z 239.088,A -85,B 0,C 180,E1 -5469.052,E2 -5469.052} C_VEL
LIN {X 0,Y 510.663,Z 256.558,A -85,B 0,C 180,E1 -5472.047,E2 -5472.047} C_VEL
LIN {X 0,Y 510.28,Z 270.687,A -85,B 0,C 180,E1 -5474.398,E2 -5474.398} C_VEL
LIN {X 0,Y 512.223,Z 283.12,A -85,B 0,C 180,E1 -5474.663,E2 -5474.663} C_VEL
LIN {X 0,Y 511.726,Z 379.172,A -85,B 0,C 180,E1 -5476.043,E2 -5476.043} C_VEL
LIN {X 0,Y 511.48,Z 392.931,A -85,B 0,C 180,E1 -5476.416,E2 -5476.416} C_VEL
LIN {X 0,Y 511.175,Z 405.786,A -85,B 0,C 180,E1 -5476.939,E2 -5476.939} C_VEL
LIN {X 0,Y 510.827,Z 418.437,A -85,B 0,C 180,E1 -5477.645,E2 -5477.645} C_VEL
LIN {X 0,Y 510.509,Z 430.112,A -85,B 0,C 180,E1 -5478.486,E2 -5478.486} C_VEL
LIN {X 0,Y 510.152,Z 441.003,A -85,B 0,C 180,E1 -5479.483,E2 -5479.483} C_VEL
LIN {X 0,Y 509.85,Z 449.849,A -85,B 0,C 180,E1 -5480.479,E2 -5480.479} C_VEL
LIN {X 0,Y 509.597,Z 458.475,A -85,B 0,C 180,E1 -5481.674,E2 -5481.674} C_VEL
LIN {X 0,Y 509.406,Z 465.364,A -85,B 0,C 180,E1 -5482.868,E2 -5482.868} C_VEL
LIN {X 0,Y 509.342,Z 470.884,A -85,B 0,C 180,E1 -5484.06,E2 -5484.06} C_VEL
LIN {X 0,Y 509.187,Z 475.211,A -85,B 0,C 180,E1 -5485.25,E2 -5485.25} C_VEL
LIN {X 0,Y 509.247,Z 477.502,A -85,B 0,C 180,E1 -5486.044,E2 -5486.044} C_VEL
LIN {X 0,Y 509.202,Z 479.358,A -85,B 0,C 180,E1 -5486.835,E2 -5486.835} C_VEL
LIN {X 0,Y 509.162,Z 480.749,A -85,B 0,C 180,E1 -5487.627,E2 -5487.627} C_VEL
LIN {X 0,Y 509.074,Z 482.346,A -85,B 0,C 180,E1 -5489.209,E2 -5489.209} C_VEL
LIN {X 0,Y 509.067,Z 482.561,A -85,B 0,C 180,E1 -5490,E2 -5490} C_VEL
LIN {X 0,Y 509.113,Z 481.739,A -85,B 0,C 180,E1 -5491.582,E2 -5491.582} C_VEL
LIN {X 0,Y 509.162,Z 480.747,A -85,B 0,C 180,E1 -5492.374,E2 -5492.374} C_VEL
LIN {X 0,Y 509.202,Z 479.354,A -85,B 0,C 180,E1 -5493.165,E2 -5493.165} C_VEL
LIN {X 0,Y 509.206,Z 476.425,A -85,B 0,C 180,E1 -5494.354,E2 -5494.354} C_VEL
LIN {X 0,Y 509.313,Z 472.46,A -85,B 0,C 180,E1 -5495.543,E2 -5495.543} C_VEL
LIN {X 0,Y 509.368,Z 466.458,A -85,B 0,C 180,E1 -5496.914,E2 -5496.914} C_VEL
LIN {X 0,Y 509.563,Z 459.689,A -85,B 0,C 180,E1 -5498.127,E2 -5498.127} C_VEL
LIN {X 0,Y 509.772,Z 451.412,A -85,B 0,C 180,E1 -5499.323,E2 -5499.323} C_VEL
LIN {X 0,Y 510.034,Z 442.923,A -85,B 0,C 180,E1 -5500.319,E2 -5500.319} C_VEL
LIN {X 0,Y 510.402,Z 432.431,A -85,B 0,C 180,E1 -5501.316,E2 -5501.316} C_VEL
LIN {X 0,Y 510.701,Z 421.938,A -85,B 0,C 180,E1 -5502.122,E2 -5502.122} C_VEL
LIN {X 0,Y 511.065,Z 410.656,A -85,B 0,C 180,E1 -5502.812,E2 -5502.812} C_VEL
LIN {X 0,Y 511.342,Z 398.934,A -85,B 0,C 180,E1 -5503.361,E2 -5503.361} C_VEL
LIN {X 0,Y 511.605,Z 385.421,A -85,B 0,C 180,E1 -5503.809,E2 -5503.809} C_VEL
LIN {X 0,Y 511.787,Z 371.909,A -85,B 0,C 180,E1 -5504.083,E2 -5504.083} C_VEL
LIN {X 0,Y 512.17,Z 282.479,A -85,B 0,C 180,E1 -5505.347,E2 -5505.347} C_VEL
LIN {X 0,Y 510.291,Z 270.756,A -85,B 0,C 180,E1 -5505.593,E2 -5505.593} C_VEL
LIN {X 0,Y 510.317,Z 266.859,A -85,B 0,C 180,E1 -5506.194,E2 -5506.194} C_VEL
LIN {X 0,Y 510.719,Z 251.052,A -85,B 0,C 180,E1 -5508.868,E2 -5508.868} C_VEL
LIN {X 0,Y 511.292,Z 232.806,A -85,B 0,C 180,E1 -5511.998,E2 -5511.998} C_VEL
LIN {X 0,Y 510.472,Z 226.67,A -85,B 0,C 180,E1 -5513.11,E2 -5513.11} C_VEL
LIN {X 0,Y 509.884,Z 223.52,A -85,B 0,C 180,E1 -5513.75,E2 -5513.75} C_VEL
LIN {X 0,Y 509.882,Z 223.471,A -85,B 0,C 180,E1 -5517.056,E2 -5517.056} C_VEL
LIN {X 0,Y 509.866,Z 223.476,A -85,B 0,C 180,E1 -5519.751,E2 -5519.751} C_VEL
LIN {X 0,Y 509.882,Z 223.466,A -85,B 0,C 180,E1 -5522.773,E2 -5522.773} C_VEL
LIN {X 0,Y 509.831,Z 223.475,A -85,B 0,C 180,E1 -5525.577,E2 -5525.577} C_VEL
LIN {X 0,Y 509.858,Z 223.474,A -85,B 0,C 180,E1 -5528.337,E2 -5528.337} C_VEL
LIN {X 0,Y 509.854,Z 223.47,A -85,B 0,C 180,E1 -5531.426,E2 -5531.426} C_VEL
LIN {X 0,Y 509.849,Z 223.477,A -85,B 0,C 180,E1 -5534.669,E2 -5534.669} C_VEL
LIN {X 0,Y 509.857,Z 223.466,A -85,B 0,C 180,E1 -5538.103,E2 -5538.103} C_VEL
LIN {X 0,Y 509.847,Z 223.479,A -85,B 0,C 180,E1 -5540.645,E2 -5540.645} C_VEL
LIN {X 0,Y 509.818,Z 223.475,A -85,B 0,C 180,E1 -5543.644,E2 -5543.644} C_VEL
LIN {X 0,Y 509.848,Z 223.476,A -85,B 0,C 180,E1 -5546.536,E2 -5546.536} C_VEL
LIN {X 0,Y 509.843,Z 223.476,A -85,B 0,C 180,E1 -5549.332,E2 -5549.332} C_VEL
LIN {X 0,Y 509.842,Z 223.469,A -85,B 0,C 180,E1 -5552.049,E2 -5552.049} C_VEL
LIN {X 0,Y 509.81,Z 223.479,A -85,B 0,C 180,E1 -5554.698,E2 -5554.698} C_VEL
LIN {X 0,Y 509.833,Z 223.479,A -85,B 0,C 180,E1 -5557.456,E2 -5557.456} C_VEL
LIN {X 0,Y 509.923,Z 223.461,A -85,B 0,C 180,E1 -5559.842,E2 -5559.842} C_VEL
LIN {X 0,Y 509.879,Z 223.472,A -85,B 0,C 180,E1 -5563.172,E2 -5563.172} C_VEL
LIN {X 0,Y 509.864,Z 223.477,A -85,B 0,C 180,E1 -5565.631,E2 -5565.631} C_VEL
LIN {X 0,Y 509.917,Z 223.46,A -85,B 0,C 180,E1 -5568.872,E2 -5568.872} C_VEL
LIN {X 0,Y 509.916,Z 223.466,A -85,B 0,C 180,E1 -5572.075,E2 -5572.075} C_VEL
LIN {X 0,Y 509.969,Z 223.456,A -85,B 0,C 180,E1 -5574.461,E2 -5574.461} C_VEL
LIN {X 0,Y 510.05,Z 223.45,A -85,B 0,C 180,E1 -5577.627,E2 -5577.627} C_VEL
LIN {X 0,Y 510.057,Z 223.451,A -85,B 0,C 180,E1 -5579.996,E2 -5579.996} C_VEL
LIN {X 0,Y 510.049,Z 223.448,A -85,B 0,C 180,E1 -5582.365,E2 -5582.365} C_VEL
LIN {X 0,Y 509.969,Z 223.457,A -85,B 0,C 180,E1 -5585.532,E2 -5585.532} C_VEL
LIN {X 0,Y 509.905,Z 223.468,A -85,B 0,C 180,E1 -5588.716,E2 -5588.716} C_VEL
LIN {X 0,Y 509.898,Z 223.463,A -85,B 0,C 180,E1 -5591.928,E2 -5591.928} C_VEL
LIN {X 0,Y 509.885,Z 223.466,A -85,B 0,C 180,E1 -5595.238,E2 -5595.238} C_VEL
LIN {X 0,Y 509.856,Z 223.471,A -85,B 0,C 180,E1 -5597.989,E2 -5597.989} C_VEL
LIN {X 0,Y 509.874,Z 223.471,A -85,B 0,C 180,E1 -5600.397,E2 -5600.397} C_VEL
LIN {X 0,Y 509.823,Z 223.475,A -85,B 0,C 180,E1 -5603.559,E2 -5603.559} C_VEL
LIN {X 0,Y 509.894,Z 223.46,A -85,B 0,C 180,E1 -5606.374,E2 -5606.374} C_VEL
LIN {X 0,Y 509.857,Z 223.476,A -85,B 0,C 180,E1 -5608.84,E2 -5608.84} C_VEL
LIN {X 0,Y 509.799,Z 223.48,A -85,B 0,C 180,E1 -5611.586,E2 -5611.586} C_VEL
LIN {X 0,Y 509.829,Z 223.473,A -85,B 0,C 180,E1 -5614.409,E2 -5614.409} C_VEL
LIN {X 0,Y 509.795,Z 223.485,A -85,B 0,C 180,E1 -5617.336,E2 -5617.336} C_VEL
LIN {X 0,Y 509.85,Z 223.471,A -85,B 0,C 180,E1 -5620.374,E2 -5620.374} C_VEL
LIN {X 0,Y 509.809,Z 223.479,A -85,B 0,C 180,E1 -5623.06,E2 -5623.06} C_VEL
LIN {X 0,Y 509.797,Z 223.486,A -85,B 0,C 180,E1 -5625.788,E2 -5625.788} C_VEL
LIN {X 0,Y 509.838,Z 223.476,A -85,B 0,C 180,E1 -5628.573,E2 -5628.573} C_VEL
LIN {X 0,Y 509.945,Z 223.647,A -85,B 0,C 180,E1 -5630.339,E2 -5630.339} C_VEL
LIN {X 0,Y 510.774,Z 229.498,A -85,B 0,C 180,E1 -5631.474,E2 -5631.474} C_VEL
LIN {X 0,Y 510.587,Z 239.154,A -85,B 0,C 180,E1 -5633.217,E2 -5633.217} C_VEL
LIN {X 0,Y 509.797,Z 242.408,A -85,B 0,C 180,E1 -5633.771,E2 -5633.771} C_VEL
LIN {X 0,Y 503.82,Z 253.354,A -85,B 0,C 180,E1 -5635.533,E2 -5635.533} C_VEL
LIN {X 0,Y 503.257,Z 256.529,A -85,B 0,C 180,E1 -5636.083,E2 -5636.083} C_VEL
LIN {X 0,Y 503.34,Z 257.919,A -85,B 0,C 180,E1 -5636.24,E2 -5636.24} C_VEL
LIN {X 0,Y 505.434,Z 269.933,A -85,B 0,C 180,E1 -5636.499,E2 -5636.499} C_VEL
LIN {X 0,Y 504.846,Z 365.158,A -85,B 0,C 180,E1 -5637.885,E2 -5637.885} C_VEL
LIN {X 0,Y 504.631,Z 378.754,A -85,B 0,C 180,E1 -5638.257,E2 -5638.257} C_VEL
LIN {X 0,Y 504.329,Z 391.749,A -85,B 0,C 180,E1 -5638.787,E2 -5638.787} C_VEL
LIN {X 0,Y 504.007,Z 402.922,A -85,B 0,C 180,E1 -5639.405,E2 -5639.405} C_VEL
LIN {X 0,Y 503.654,Z 414.07,A -85,B 0,C 180,E1 -5640.191,E2 -5640.191} C_VEL
LIN {X 0,Y 503.285,Z 424.276,A -85,B 0,C 180,E1 -5641.085,E2 -5641.085} C_VEL
LIN {X 0,Y 502.991,Z 433.584,A -85,B 0,C 180,E1 -5642.09,E2 -5642.09} C_VEL
LIN {X 0,Y 502.657,Z 441.924,A -85,B 0,C 180,E1 -5643.198,E2 -5643.198} C_VEL
LIN {X 0,Y 502.432,Z 449.958,A -85,B 0,C 180,E1 -5644.524,E2 -5644.524} C_VEL
LIN {X 0,Y 502.283,Z 455.788,A -85,B 0,C 180,E1 -5645.737,E2 -5645.737} C_VEL
LIN {X 0,Y 502.156,Z 460.307,A -85,B 0,C 180,E1 -5646.928,E2 -5646.928} C_VEL
LIN {X 0,Y 502.091,Z 464.03,A -85,B 0,C 180,E1 -5648.227,E2 -5648.227} C_VEL
LIN {X 0,Y 502.057,Z 466.819,A -85,B 0,C 180,E1 -5649.683,E2 -5649.683} C_VEL
LIN {X 0,Y 501.974,Z 468.327,A -85,B 0,C 180,E1 -5651.215,E2 -5651.215} C_VEL
LIN {X 0,Y 501.984,Z 468.54,A -85,B 0,C 180,E1 -5652.161,E2 -5652.161} C_VEL
LIN {X 0,Y 502.009,Z 467.646,A -85,B 0,C 180,E1 -5653.74,E2 -5653.74} C_VEL
LIN {X 0,Y 502.092,Z 465.912,A -85,B 0,C 180,E1 -5654.953,E2 -5654.953} C_VEL
LIN {X 0,Y 502.128,Z 461.899,A -85,B 0,C 180,E1 -5656.647,E2 -5656.647} C_VEL
LIN {X 0,Y 502.221,Z 457.675,A -85,B 0,C 180,E1 -5657.883,E2 -5657.883} C_VEL
LIN {X 0,Y 502.365,Z 452.256,A -85,B 0,C 180,E1 -5659.113,E2 -5659.113} C_VEL
LIN {X 0,Y 502.548,Z 445.485,A -85,B 0,C 180,E1 -5660.339,E2 -5660.339} C_VEL
LIN {X 0,Y 502.876,Z 437.079,A -85,B 0,C 180,E1 -5661.561,E2 -5661.561} C_VEL
LIN {X 0,Y 503.169,Z 427.577,A -85,B 0,C 180,E1 -5662.667,E2 -5662.667} C_VEL
LIN {X 0,Y 503.506,Z 417.838,A -85,B 0,C 180,E1 -5663.588,E2 -5663.588} C_VEL
LIN {X 0,Y 503.853,Z 407.316,A -85,B 0,C 180,E1 -5664.396,E2 -5664.396} C_VEL
LIN {X 0,Y 504.231,Z 395.64,A -85,B 0,C 180,E1 -5665.102,E2 -5665.102} C_VEL
LIN {X 0,Y 504.522,Z 383.548,A -85,B 0,C 180,E1 -5665.656,E2 -5665.656} C_VEL
LIN {X 0,Y 504.729,Z 370.403,A -85,B 0,C 180,E1 -5666.082,E2 -5666.082} C_VEL
LIN {X 0,Y 504.928,Z 357.393,A -85,B 0,C 180,E1 -5666.334,E2 -5666.334} C_VEL
LIN {X 0,Y 505.264,Z 268.621,A -85,B 0,C 180,E1 -5667.608,E2 -5667.608} C_VEL
LIN {X 0,Y 503.33,Z 257.752,A -85,B 0,C 180,E1 -5667.849,E2 -5667.849} C_VEL
LIN {X 0,Y 503.315,Z 254.483,A -85,B 0,C 180,E1 -5668.399,E2 -5668.399} C_VEL
LIN {X 0,Y 503.73,Z 239.544,A -85,B 0,C 180,E1 -5671.199,E2 -5671.199} C_VEL
LIN {X 0,Y 504.044,Z 231.073,A -85,B 0,C 180,E1 -5672.797,E2 -5672.797} C_VEL
LIN {X 0,Y 502.811,Z 224.457,A -85,B 0,C 180,E1 -5674.158,E2 -5674.158} C_VEL
LIN {X 0,Y 502.942,Z 224.34,A -85,B 0,C 180,E1 -5676.418,E2 -5676.418} C_VEL
LIN {X 0,Y 502.869,Z 224.346,A -85,B 0,C 180,E1 -5678.843,E2 -5678.843} C_VEL
LIN {X 0,Y 502.851,Z 224.346,A -85,B 0,C 180,E1 -5682.101,E2 -5682.101} C_VEL
LIN {X 0,Y 502.833,Z 224.346,A -85,B 0,C 180,E1 -5685.4,E2 -5685.4} C_VEL
LIN {X 0,Y 502.815,Z 224.346,A -85,B 0,C 180,E1 -5688.131,E2 -5688.131} C_VEL
LIN {X 0,Y 502.788,Z 224.354,A -85,B 0,C 180,E1 -5691.311,E2 -5691.311} C_VEL
LIN {X 0,Y 502.782,Z 224.35,A -85,B 0,C 180,E1 -5693.914,E2 -5693.914} C_VEL
LIN {X 0,Y 502.834,Z 224.336,A -85,B 0,C 180,E1 -5696.567,E2 -5696.567} C_VEL
LIN {X 0,Y 502.807,Z 224.35,A -85,B 0,C 180,E1 -5699.288,E2 -5699.288} C_VEL
LIN {X 0,Y 502.766,Z 224.355,A -85,B 0,C 180,E1 -5702.085,E2 -5702.085} C_VEL
LIN {X 0,Y 502.799,Z 224.348,A -85,B 0,C 180,E1 -5704.965,E2 -5704.965} C_VEL
LIN {X 0,Y 502.778,Z 224.352,A -85,B 0,C 180,E1 -5708.493,E2 -5708.493} C_VEL
LIN {X 0,Y 502.795,Z 224.348,A -85,B 0,C 180,E1 -5711.068,E2 -5711.068} C_VEL
LIN {X 0,Y 502.793,Z 224.351,A -85,B 0,C 180,E1 -5714.338,E2 -5714.338} C_VEL
LIN {X 0,Y 502.792,Z 224.35,A -85,B 0,C 180,E1 -5716.778,E2 -5716.778} C_VEL
LIN {X 0,Y 502.803,Z 224.351,A -85,B 0,C 180,E1 -5719.993,E2 -5719.993} C_VEL
LIN {X 0,Y 502.755,Z 224.35,A -85,B 0,C 180,E1 -5723.058,E2 -5723.058} C_VEL
LIN {X 0,Y 502.786,Z 224.354,A -85,B 0,C 180,E1 -5726.011,E2 -5726.011} C_VEL
LIN {X 0,Y 502.774,Z 224.352,A -85,B 0,C 180,E1 -5728.861,E2 -5728.861} C_VEL
LIN {X 0,Y 502.823,Z 224.336,A -85,B 0,C 180,E1 -5731.708,E2 -5731.708} C_VEL
LIN {X 0,Y 502.822,Z 224.342,A -85,B 0,C 180,E1 -5734.329,E2 -5734.329} C_VEL
LIN {X 0,Y 502.789,Z 224.352,A -85,B 0,C 180,E1 -5737.3,E2 -5737.3} C_VEL
LIN {X 0,Y 502.811,Z 224.349,A -85,B 0,C 180,E1 -5740.404,E2 -5740.404} C_VEL
LIN {X 0,Y 502.823,Z 224.345,A -85,B 0,C 180,E1 -5742.936,E2 -5742.936} C_VEL
LIN {X 0,Y 502.832,Z 224.339,A -85,B 0,C 180,E1 -5745.433,E2 -5745.433} C_VEL
LIN {X 0,Y 502.886,Z 224.336,A -85,B 0,C 180,E1 -5748.721,E2 -5748.721} C_VEL
LIN {X 0,Y 502.895,Z 224.337,A -85,B 0,C 180,E1 -5751.971,E2 -5751.971} C_VEL
LIN {X 0,Y 502.935,Z 224.328,A -85,B 0,C 180,E1 -5754.39,E2 -5754.39} C_VEL
LIN {X 0,Y 503.02,Z 224.315,A -85,B 0,C 180,E1 -5757.601,E2 -5757.601} C_VEL
LIN {X 0,Y 503.024,Z 224.32,A -85,B 0,C 180,E1 -5760.004,E2 -5760.004} C_VEL
LIN {X 0,Y 503.023,Z 224.321,A -85,B 0,C 180,E1 -5762.406,E2 -5762.406} C_VEL
LIN {X 0,Y 502.928,Z 224.337,A -85,B 0,C 180,E1 -5765.617,E2 -5765.617} C_VEL
LIN {X 0,Y 502.87,Z 224.331,A -85,B 0,C 180,E1 -5768.847,E2 -5768.847} C_VEL
LIN {X 0,Y 502.848,Z 224.342,A -85,B 0,C 180,E1 -5772.105,E2 -5772.105} C_VEL
LIN {X 0,Y 502.852,Z 224.342,A -85,B 0,C 180,E1 -5775.403,E2 -5775.403} C_VEL
LIN {X 0,Y 502.83,Z 224.344,A -85,B 0,C 180,E1 -5778.755,E2 -5778.755} C_VEL
LIN {X 0,Y 502.788,Z 224.343,A -85,B 0,C 180,E1 -5781.314,E2 -5781.314} C_VEL
LIN {X 0,Y 502.786,Z 224.349,A -85,B 0,C 180,E1 -5783.917,E2 -5783.917} C_VEL
LIN {X 0,Y 502.841,Z 224.351,A -85,B 0,C 180,E1 -5786.57,E2 -5786.57} C_VEL
LIN {X 0,Y 502.828,Z 224.341,A -85,B 0,C 180,E1 -5789.29,E2 -5789.29} C_VEL
LIN {X 0,Y 502.788,Z 224.349,A -85,B 0,C 180,E1 -5792.087,E2 -5792.087} C_VEL
LIN {X 0,Y 502.8,Z 224.358,A -85,B 0,C 180,E1 -5794.968,E2 -5794.968} C_VEL
LIN {X 0,Y 502.8,Z 224.347,A -85,B 0,C 180,E1 -5798.488,E2 -5798.488} C_VEL
LIN {X 0,Y 502.807,Z 224.354,A -85,B 0,C 180,E1 -5801.07,E2 -5801.07} C_VEL
LIN {X 0,Y 502.786,Z 224.339,A -85,B 0,C 180,E1 -5804.342,E2 -5804.342} C_VEL
LIN {X 0,Y 502.761,Z 224.347,A -85,B 0,C 180,E1 -5806.768,E2 -5806.768} C_VEL
LIN {X 0,Y 502.806,Z 224.349,A -85,B 0,C 180,E1 -5809.009,E2 -5809.009} C_VEL
LIN {X 0,Y 502.797,Z 224.353,A -85,B 0,C 180,E1 -5812.047,E2 -5812.047} C_VEL
LIN {X 0,Y 502.804,Z 224.348,A -85,B 0,C 180,E1 -5815.035,E2 -5815.035} C_VEL
LIN {X 0,Y 502.79,Z 224.358,A -85,B 0,C 180,E1 -5817.916,E2 -5817.916} C_VEL
LIN {X 0,Y 502.829,Z 224.349,A -85,B 0,C 180,E1 -5820.713,E2 -5820.713} C_VEL
LIN {X 0,Y 502.853,Z 224.346,A -85,B 0,C 180,E1 -5823.444,E2 -5823.444} C_VEL
LIN {X 0,Y 502.848,Z 224.506,A -85,B 0,C 180,E1 -5826.09,E2 -5826.09} C_VEL
LIN {X 0,Y 504.332,Z 232.909,A -85,B 0,C 180,E1 -5827.683,E2 -5827.683} C_VEL
LIN {X 0,Y 503.887,Z 248.677,A -85,B 0,C 180,E1 -5830.444,E2 -5830.444} C_VEL
LIN {X 0,Y 503.437,Z 263.208,A -85,B 0,C 180,E1 -5832.953,E2 -5832.953} C_VEL
LIN {X 0,Y 503.282,Z 270.517,A -85,B 0,C 180,E1 -5834.174,E2 -5834.174} C_VEL
LIN {X 0,Y 504.619,Z 278.789,A -85,B 0,C 180,E1 -5834.367,E2 -5834.367} C_VEL
LIN {X 0,Y 505.395,Z 284.525,A -85,B 0,C 180,E1 -5834.474,E2 -5834.474} C_VEL
LIN {X 0,Y 504.848,Z 379.021,A -85,B 0,C 180,E1 -5835.849,E2 -5835.849} C_VEL
LIN {X 0,Y 504.593,Z 392.797,A -85,B 0,C 180,E1 -5836.227,E2 -5836.227} C_VEL
LIN {X 0,Y 504.245,Z 405.664,A -85,B 0,C 180,E1 -5836.756,E2 -5836.756} C_VEL
LIN {X 0,Y 503.895,Z 418.093,A -85,B 0,C 180,E1 -5837.457,E2 -5837.457} C_VEL
LIN {X 0,Y 503.596,Z 428.731,A -85,B 0,C 180,E1 -5838.223,E2 -5838.223} C_VEL
LIN {X 0,Y 503.183,Z 438.936,A -85,B 0,C 180,E1 -5839.132,E2 -5839.132} C_VEL
LIN {X 0,Y 502.875,Z 448.111,A -85,B 0,C 180,E1 -5840.143,E2 -5840.143} C_VEL
LIN {X 0,Y 502.6,Z 457.047,A -85,B 0,C 180,E1 -5841.355,E2 -5841.355} C_VEL
LIN {X 0,Y 502.36,Z 464.237,A -85,B 0,C 180,E1 -5842.565,E2 -5842.565} C_VEL
LIN {X 0,Y 502.241,Z 469.088,A -85,B 0,C 180,E1 -5843.573,E2 -5843.573} C_VEL
LIN {X 0,Y 502.181,Z 473.802,A -85,B 0,C 180,E1 -5844.781,E2 -5844.781} C_VEL
LIN {X 0,Y 502.14,Z 477.402,A -85,B 0,C 180,E1 -5845.987,E2 -5845.987} C_VEL
LIN {X 0,Y 502.122,Z 479.259,A -85,B 0,C 180,E1 -5846.791,E2 -5846.791} C_VEL
LIN {X 0,Y 502.037,Z 481.643,A -85,B 0,C 180,E1 -5848.396,E2 -5848.396} C_VEL
LIN {X 0,Y 501.982,Z 482.463,A -85,B 0,C 180,E1 -5850,E2 -5850} C_VEL
LIN {X 0,Y 502.037,Z 481.641,A -85,B 0,C 180,E1 -5851.605,E2 -5851.605} C_VEL
LIN {X 0,Y 502.067,Z 480.647,A -85,B 0,C 180,E1 -5852.407,E2 -5852.407} C_VEL
LIN {X 0,Y 502.122,Z 479.254,A -85,B 0,C 180,E1 -5853.21,E2 -5853.21} C_VEL
LIN {X 0,Y 502.104,Z 476.323,A -85,B 0,C 180,E1 -5854.415,E2 -5854.415} C_VEL
LIN {X 0,Y 502.231,Z 472.357,A -85,B 0,C 180,E1 -5855.622,E2 -5855.622} C_VEL
LIN {X 0,Y 502.294,Z 466.353,A -85,B 0,C 180,E1 -5857.012,E2 -5857.012} C_VEL
LIN {X 0,Y 502.495,Z 459.581,A -85,B 0,C 180,E1 -5858.242,E2 -5858.242} C_VEL
LIN {X 0,Y 502.744,Z 451.302,A -85,B 0,C 180,E1 -5859.454,E2 -5859.454} C_VEL
LIN {X 0,Y 503.02,Z 442.81,A -85,B 0,C 180,E1 -5860.465,E2 -5860.465} C_VEL
LIN {X 0,Y 503.443,Z 432.315,A -85,B 0,C 180,E1 -5861.474,E2 -5861.474} C_VEL
LIN {X 0,Y 503.72,Z 421.816,A -85,B 0,C 180,E1 -5862.293,E2 -5862.293} C_VEL
LIN {X 0,Y 504.124,Z 410.538,A -85,B 0,C 180,E1 -5862.991,E2 -5862.991} C_VEL
LIN {X 0,Y 504.441,Z 398.822,A -85,B 0,C 180,E1 -5863.547,E2 -5863.547} C_VEL
LIN {X 0,Y 504.735,Z 385.322,A -85,B 0,C 180,E1 -5864.001,E2 -5864.001} C_VEL
LIN {X 0,Y 504.928,Z 371.836,A -85,B 0,C 180,E1 -5864.278,E2 -5864.278} C_VEL
LIN {X 0,Y 505.308,Z 283.085,A -85,B 0,C 180,E1 -5865.553,E2 -5865.553} C_VEL
LIN {X 0,Y 503.315,Z 270.634,A -85,B 0,C 180,E1 -5865.824,E2 -5865.824} C_VEL
LIN {X 0,Y 503.338,Z 266.788,A -85,B 0,C 180,E1 -5866.424,E2 -5866.424} C_VEL
LIN {X 0,Y 503.782,Z 250.973,A -85,B 0,C 180,E1 -5869.138,E2 -5869.138} C_VEL
LIN {X 0,Y 504.362,Z 233.959,A -85,B 0,C 180,E1 -5872.1,E2 -5872.1} C_VEL
LIN {X 0,Y 503.276,Z 226.674,A -85,B 0,C 180,E1 -5873.453,E2 -5873.453} C_VEL
LIN {X 0,Y 502.862,Z 224.406,A -85,B 0,C 180,E1 -5873.938,E2 -5873.938} C_VEL
LIN {X 0,Y 502.832,Z 224.352,A -85,B 0,C 180,E1 -5877.467,E2 -5877.467} C_VEL
LIN {X 0,Y 502.817,Z 224.351,A -85,B 0,C 180,E1 -5880.211,E2 -5880.211} C_VEL
LIN {X 0,Y 502.842,Z 224.342,A -85,B 0,C 180,E1 -5883.031,E2 -5883.031} C_VEL
LIN {X 0,Y 502.777,Z 224.356,A -85,B 0,C 180,E1 -5885.951,E2 -5885.951} C_VEL
LIN {X 0,Y 502.803,Z 224.347,A -85,B 0,C 180,E1 -5888.976,E2 -5888.976} C_VEL
LIN {X 0,Y 502.814,Z 224.351,A -85,B 0,C 180,E1 -5892.198,E2 -5892.198} C_VEL
LIN {X 0,Y 502.796,Z 224.35,A -85,B 0,C 180,E1 -5895.469,E2 -5895.469} C_VEL
LIN {X 0,Y 502.806,Z 224.342,A -85,B 0,C 180,E1 -5897.859,E2 -5897.859} C_VEL
LIN {X 0,Y 502.806,Z 224.351,A -85,B 0,C 180,E1 -5901.022,E2 -5901.022} C_VEL
LIN {X 0,Y 502.78,Z 224.353,A -85,B 0,C 180,E1 -5904.168,E2 -5904.168} C_VEL
LIN {X 0,Y 502.813,Z 224.353,A -85,B 0,C 180,E1 -5906.997,E2 -5906.997} C_VEL
LIN {X 0,Y 502.82,Z 224.347,A -85,B 0,C 180,E1 -5910.064,E2 -5910.064} C_VEL
LIN {X 0,Y 502.784,Z 224.355,A -85,B 0,C 180,E1 -5913.458,E2 -5913.458} C_VEL
LIN {X 0,Y 502.774,Z 224.35,A -85,B 0,C 180,E1 -5916.083,E2 -5916.083} C_VEL
LIN {X 0,Y 502.788,Z 224.352,A -85,B 0,C 180,E1 -5918.686,E2 -5918.686} C_VEL
LIN {X 0,Y 502.833,Z 224.349,A -85,B 0,C 180,E1 -5921.245,E2 -5921.245} C_VEL
LIN {X 0,Y 502.856,Z 224.338,A -85,B 0,C 180,E1 -5924.598,E2 -5924.598} C_VEL
LIN {X 0,Y 502.883,Z 224.339,A -85,B 0,C 180,E1 -5928.036,E2 -5928.036} C_VEL
LIN {X 0,Y 502.854,Z 224.343,A -85,B 0,C 180,E1 -5931.153,E2 -5931.153} C_VEL
LIN {X 0,Y 502.895,Z 224.342,A -85,B 0,C 180,E1 -5933.578,E2 -5933.578} C_VEL
LIN {X 0,Y 502.862,Z 224.341,A -85,B 0,C 180,E1 -5936.792,E2 -5936.792} C_VEL
LIN {X 0,Y 502.895,Z 224.338,A -85,B 0,C 180,E1 -5938.395,E2 -5938.395} C_VEL
LIN {X 0,Y 502.989,Z 224.326,A -85,B 0,C 180,E1 -5940.797,E2 -5940.797} C_VEL
LIN {X 0,Y 503.017,Z 224.323,A -85,B 0,C 180,E1 -5942.399,E2 -5942.399} C_VEL
LIN {X 0,Y 502.923,Z 224.335,A -85,B 0,C 180,E1 -5945.61,E2 -5945.61} C_VEL
LIN {X 0,Y 502.864,Z 224.344,A -85,B 0,C 180,E1 -5948.839,E2 -5948.839} C_VEL
LIN {X 0,Y 502.839,Z 224.344,A -85,B 0,C 180,E1 -5952.098,E2 -5952.098} C_VEL
LIN {X 0,Y 502.84,Z 224.342,A -85,B 0,C 180,E1 -5955.396,E2 -5955.396} C_VEL
LIN {X 0,Y 502.815,Z 224.353,A -85,B 0,C 180,E1 -5958.748,E2 -5958.748} C_VEL
LIN {X 0,Y 502.773,Z 224.353,A -85,B 0,C 180,E1 -5961.307,E2 -5961.307} C_VEL
LIN {X 0,Y 502.777,Z 224.352,A -85,B 0,C 180,E1 -5963.909,E2 -5963.909} C_VEL
LIN {X 0,Y 502.846,Z 224.34,A -85,B 0,C 180,E1 -5966.562,E2 -5966.562} C_VEL
LIN {X 0,Y 502.804,Z 224.353,A -85,B 0,C 180,E1 -5969.283,E2 -5969.283} C_VEL
LIN {X 0,Y 502.762,Z 224.353,A -85,B 0,C 180,E1 -5972.08,E2 -5972.08} C_VEL
LIN {X 0,Y 502.784,Z 224.354,A -85,B 0,C 180,E1 -5974.961,E2 -5974.961} C_VEL
LIN {X 0,Y 502.772,Z 224.352,A -85,B 0,C 180,E1 -5977.949,E2 -5977.949} C_VEL
LIN {X 0,Y 502.802,Z 224.352,A -85,B 0,C 180,E1 -5981.061,E2 -5981.061} C_VEL
LIN {X 0,Y 502.751,Z 224.361,A -85,B 0,C 180,E1 -5983.372,E2 -5983.372} C_VEL
LIN {X 0,Y 502.757,Z 224.363,A -85,B 0,C 180,E1 -5985.657,E2 -5985.657} C_VEL
LIN {X 0,Y 502.804,Z 224.356,A -85,B 0,C 180,E1 -5987.861,E2 -5987.861} C_VEL
LIN {X 0,Y 502.868,Z 224.445,A -85,B 0,C 180,E1 -5990.144,E2 -5990.144} C_VEL
LIN {X 0,Y 503.816,Z 230.544,A -85,B 0,C 180,E1 -5991.359,E2 -5991.359} C_VEL
LIN {X 0,Y 503.554,Z 245.597,A -85,B 0,C 180,E1 -5994.113,E2 -5994.113} C_VEL
LIN {X 0,Y 503.257,Z 256.529,A -85,B 0,C 180,E1 -5996.083,E2 -5996.083} C_VEL
LIN {X 0,Y 502.902,Z 258.168,A -85,B 0,C 180,E1 -5996.213,E2 -5996.213} C_VEL
LIN {X 0,Y 501.719,Z 261.03,A -85,B 0,C 180,E1 -5996.244,E2 -5996.244} C_VEL
LIN {X 0,Y 498.995,Z 268.468,A -85,B 0,C 180,E1 -5996.264,E2 -5996.264} C_VEL
LIN {X 0,Y 498.144,Z 272.575,A -85,B 0,C 180,E1 -5996.276,E2 -5996.276} C_VEL
LIN {X 0,Y 498.049,Z 279.039,A -85,B 0,C 180,E1 -5996.363,E2 -5996.363} C_VEL
LIN {X 0,Y 498.518,Z 287.706,A -85,B 0,C 180,E1 -5996.535,E2 -5996.535} C_VEL
LIN {X 0,Y 497.985,Z 364.781,A -85,B 0,C 180,E1 -5997.673,E2 -5997.673} C_VEL
LIN {X 0,Y 497.732,Z 378.414,A -85,B 0,C 180,E1 -5998.044,E2 -5998.044} C_VEL
LIN {X 0,Y 497.434,Z 390.708,A -85,B 0,C 180,E1 -5998.542,E2 -5998.542} C_VEL
LIN {X 0,Y 497.101,Z 402.194,A -85,B 0,C 180,E1 -5999.169,E2 -5999.169} C_VEL
LIN {X 0,Y 496.713,Z 413.916,A -85,B 0,C 180,E1 -6000,E2 -6000} C_VEL
LIN {X 0,Y 496.277,Z 424.984,A -85,B 0,C 180,E1 -6000.985,E2 -6000.985} C_VEL
LIN {X 0,Y 495.987,Z 433.38,A -85,B 0,C 180,E1 -6001.909,E2 -6001.909} C_VEL
LIN {X 0,Y 495.651,Z 441.664,A -85,B 0,C 180,E1 -6003.016,E2 -6003.016} C_VEL
LIN {X 0,Y 495.377,Z 449.754,A -85,B 0,C 180,E1 -6004.36,E2 -6004.36} C_VEL
LIN {X 0,Y 495.22,Z 456.099,A -85,B 0,C 180,E1 -6005.697,E2 -6005.697} C_VEL
LIN {X 0,Y 495.058,Z 460.835,A -85,B 0,C 180,E1 -6006.991,E2 -6006.991} C_VEL
LIN {X 0,Y 494.983,Z 464.489,A -85,B 0,C 180,E1 -6008.336,E2 -6008.336} C_VEL
LIN {X 0,Y 494.974,Z 466.788,A -85,B 0,C 180,E1 -6009.555,E2 -6009.555} C_VEL
LIN {X 0,Y 494.911,Z 468.268,A -85,B 0,C 180,E1 -6010.937,E2 -6010.937} C_VEL
LIN {X 0,Y 494.897,Z 468.654,A -85,B 0,C 180,E1 -6012.055,E2 -6012.055} C_VEL
LIN {X 0,Y 494.901,Z 468.004,A -85,B 0,C 180,E1 -6013.5,E2 -6013.5} C_VEL
LIN {X 0,Y 494.989,Z 466.216,A -85,B 0,C 180,E1 -6014.878,E2 -6014.878} C_VEL
LIN {X 0,Y 495.026,Z 462.735,A -85,B 0,C 180,E1 -6016.452,E2 -6016.452} C_VEL
LIN {X 0,Y 495.112,Z 458.751,A -85,B 0,C 180,E1 -6017.706,E2 -6017.706} C_VEL
LIN {X 0,Y 495.3,Z 452.602,A -85,B 0,C 180,E1 -6019.163,E2 -6019.163} C_VEL
LIN {X 0,Y 495.509,Z 445.878,A -85,B 0,C 180,E1 -6020.406,E2 -6020.406} C_VEL
LIN {X 0,Y 495.835,Z 437.541,A -85,B 0,C 180,E1 -6021.646,E2 -6021.646} C_VEL
LIN {X 0,Y 496.146,Z 428.998,A -85,B 0,C 180,E1 -6022.675,E2 -6022.675} C_VEL
LIN {X 0,Y 496.531,Z 418.465,A -85,B 0,C 180,E1 -6023.702,E2 -6023.702} C_VEL
LIN {X 0,Y 496.896,Z 408.047,A -85,B 0,C 180,E1 -6024.521,E2 -6024.521} C_VEL
LIN {X 0,Y 497.279,Z 396.604,A -85,B 0,C 180,E1 -6025.237,E2 -6025.237} C_VEL
LIN {X 0,Y 497.594,Z 384.782,A -85,B 0,C 180,E1 -6025.798,E2 -6025.798} C_VEL
LIN {X 0,Y 497.82,Z 372.09,A -85,B 0,C 180,E1 -6026.231,E2 -6026.231} C_VEL
LIN {X 0,Y 498.04,Z 358.819,A -85,B 0,C 180,E1 -6026.511,E2 -6026.511} C_VEL
LIN {X 0,Y 498.451,Z 269.738,A -85,B 0,C 180,E1 -6027.803,E2 -6027.803} C_VEL
LIN {X 0,Y 496.31,Z 257.835,A -85,B 0,C 180,E1 -6028.072,E2 -6028.072} C_VEL
LIN {X 0,Y 496.392,Z 252.682,A -85,B 0,C 180,E1 -6028.986,E2 -6028.986} C_VEL
LIN {X 0,Y 496.917,Z 236.681,A -85,B 0,C 180,E1 -6032.026,E2 -6032.026} C_VEL
LIN {X 0,Y 496.946,Z 231.415,A -85,B 0,C 180,E1 -6033.04,E2 -6033.04} C_VEL
LIN {X 0,Y 495.798,Z 225.325,A -85,B 0,C 180,E1 -6034.318,E2 -6034.318} C_VEL
LIN {X 0,Y 495.891,Z 225.218,A -85,B 0,C 180,E1 -6036.51,E2 -6036.51} C_VEL
LIN {X 0,Y 495.831,Z 225.221,A -85,B 0,C 180,E1 -6038.97,E2 -6038.97} C_VEL
LIN {X 0,Y 495.809,Z 225.225,A -85,B 0,C 180,E1 -6042.276,E2 -6042.276} C_VEL
LIN {X 0,Y 495.804,Z 225.221,A -85,B 0,C 180,E1 -6045.466,E2 -6045.466} C_VEL
LIN {X 0,Y 495.781,Z 225.223,A -85,B 0,C 180,E1 -6048.258,E2 -6048.258} C_VEL
LIN {X 0,Y 495.749,Z 225.228,A -85,B 0,C 180,E1 -6051.628,E2 -6051.628} C_VEL
LIN {X 0,Y 495.733,Z 225.228,A -85,B 0,C 180,E1 -6054.276,E2 -6054.276} C_VEL
LIN {X 0,Y 495.776,Z 225.216,A -85,B 0,C 180,E1 -6056.976,E2 -6056.976} C_VEL
LIN {X 0,Y 495.751,Z 225.226,A -85,B 0,C 180,E1 -6060.156,E2 -6060.156} C_VEL
LIN {X 0,Y 495.771,Z 225.232,A -85,B 0,C 180,E1 -6063.251,E2 -6063.251} C_VEL
LIN {X 0,Y 495.714,Z 225.231,A -85,B 0,C 180,E1 -6066.097,E2 -6066.097} C_VEL
LIN {X 0,Y 495.772,Z 225.233,A -85,B 0,C 180,E1 -6069.636,E2 -6069.636} C_VEL
LIN {X 0,Y 495.751,Z 225.22,A -85,B 0,C 180,E1 -6072.88,E2 -6072.88} C_VEL
LIN {X 0,Y 495.76,Z 225.23,A -85,B 0,C 180,E1 -6076.301,E2 -6076.301} C_VEL
LIN {X 0,Y 495.754,Z 225.224,A -85,B 0,C 180,E1 -6079.306,E2 -6079.306} C_VEL
LIN {X 0,Y 495.708,Z 225.233,A -85,B 0,C 180,E1 -6082.443,E2 -6082.443} C_VEL
LIN {X 0,Y 495.763,Z 225.225,A -85,B 0,C 180,E1 -6085.462,E2 -6085.462} C_VEL
LIN {X 0,Y 495.735,Z 225.236,A -85,B 0,C 180,E1 -6088.368,E2 -6088.368} C_VEL
LIN {X 0,Y 495.768,Z 225.214,A -85,B 0,C 180,E1 -6091.51,E2 -6091.51} C_VEL
LIN {X 0,Y 495.779,Z 225.215,A -85,B 0,C 180,E1 -6093.937,E2 -6093.937} C_VEL
LIN {X 0,Y 495.747,Z 225.231,A -85,B 0,C 180,E1 -6097.142,E2 -6097.142} C_VEL
LIN {X 0,Y 495.762,Z 225.225,A -85,B 0,C 180,E1 -6100.114,E2 -6100.114} C_VEL
LIN {X 0,Y 495.775,Z 225.223,A -85,B 0,C 180,E1 -6102.686,E2 -6102.686} C_VEL
LIN {X 0,Y 495.777,Z 225.217,A -85,B 0,C 180,E1 -6105.221,E2 -6105.221} C_VEL
LIN {X 0,Y 495.86,Z 225.21,A -85,B 0,C 180,E1 -6108.559,E2 -6108.559} C_VEL
LIN {X 0,Y 495.866,Z 225.214,A -85,B 0,C 180,E1 -6111.856,E2 -6111.856} C_VEL
LIN {X 0,Y 495.893,Z 225.205,A -85,B 0,C 180,E1 -6114.31,E2 -6114.31} C_VEL
LIN {X 0,Y 495.988,Z 225.19,A -85,B 0,C 180,E1 -6117.567,E2 -6117.567} C_VEL
LIN {X 0,Y 495.98,Z 225.193,A -85,B 0,C 180,E1 -6120.816,E2 -6120.816} C_VEL
LIN {X 0,Y 495.991,Z 225.197,A -85,B 0,C 180,E1 -6122.44,E2 -6122.44} C_VEL
LIN {X 0,Y 495.883,Z 225.216,A -85,B 0,C 180,E1 -6125.697,E2 -6125.697} C_VEL
LIN {X 0,Y 495.839,Z 225.206,A -85,B 0,C 180,E1 -6128.973,E2 -6128.973} C_VEL
LIN {X 0,Y 495.83,Z 225.215,A -85,B 0,C 180,E1 -6132.038,E2 -6132.038} C_VEL
LIN {X 0,Y 495.827,Z 225.217,A -85,B 0,C 180,E1 -6135.455,E2 -6135.455} C_VEL
LIN {X 0,Y 495.783,Z 225.229,A -85,B 0,C 180,E1 -6138.24,E2 -6138.24} C_VEL
LIN {X 0,Y 495.779,Z 225.22,A -85,B 0,C 180,E1 -6140.759,E2 -6140.759} C_VEL
LIN {X 0,Y 495.751,Z 225.225,A -85,B 0,C 180,E1 -6143.39,E2 -6143.39} C_VEL
LIN {X 0,Y 495.81,Z 225.228,A -85,B 0,C 180,E1 -6146.747,E2 -6146.747} C_VEL
LIN {X 0,Y 495.771,Z 225.217,A -85,B 0,C 180,E1 -6149.749,E2 -6149.749} C_VEL
LIN {X 0,Y 495.758,Z 225.229,A -85,B 0,C 180,E1 -6152.598,E2 -6152.598} C_VEL
LIN {X 0,Y 495.75,Z 225.228,A -85,B 0,C 180,E1 -6155.54,E2 -6155.54} C_VEL
LIN {X 0,Y 495.769,Z 225.225,A -85,B 0,C 180,E1 -6158.77,E2 -6158.77} C_VEL
LIN {X 0,Y 495.758,Z 225.226,A -85,B 0,C 180,E1 -6161.783,E2 -6161.783} C_VEL
LIN {X 0,Y 495.744,Z 225.22,A -85,B 0,C 180,E1 -6165.143,E2 -6165.143} C_VEL
LIN {X 0,Y 495.758,Z 225.227,A -85,B 0,C 180,E1 -6168.22,E2 -6168.22} C_VEL
LIN {X 0,Y 495.753,Z 225.23,A -85,B 0,C 180,E1 -6171.409,E2 -6171.409} C_VEL
LIN {X 0,Y 495.752,Z 225.228,A -85,B 0,C 180,E1 -6174.463,E2 -6174.463} C_VEL
LIN {X 0,Y 495.775,Z 225.227,A -85,B 0,C 180,E1 -6177.407,E2 -6177.407} C_VEL
LIN {X 0,Y 495.772,Z 225.231,A -85,B 0,C 180,E1 -6180.255,E2 -6180.255} C_VEL
LIN {X 0,Y 495.813,Z 225.223,A -85,B 0,C 180,E1 -6183.256,E2 -6183.256} C_VEL
LIN {X 0,Y 495.834,Z 225.325,A -85,B 0,C 180,E1 -6185.897,E2 -6185.897} C_VEL
LIN {X 0,Y 497.353,Z 233.965,A -85,B 0,C 180,E1 -6187.572,E2 -6187.572} C_VEL
LIN {X 0,Y 496.962,Z 247.33,A -85,B 0,C 180,E1 -6189.944,E2 -6189.944} C_VEL
LIN {X 0,Y 496.474,Z 263.085,A -85,B 0,C 180,E1 -6192.707,E2 -6192.707} C_VEL
LIN {X 0,Y 496.292,Z 270.447,A -85,B 0,C 180,E1 -6193.954,E2 -6193.954} C_VEL
LIN {X 0,Y 498.423,Z 283.75,A -85,B 0,C 180,E1 -6194.246,E2 -6194.246} C_VEL
LIN {X 0,Y 497.983,Z 378.699,A -85,B 0,C 180,E1 -6195.65,E2 -6195.65} C_VEL
LIN {X 0,Y 497.726,Z 391.794,A -85,B 0,C 180,E1 -6196.007,E2 -6196.007} C_VEL
LIN {X 0,Y 497.368,Z 404.43,A -85,B 0,C 180,E1 -6196.518,E2 -6196.518} C_VEL
LIN {X 0,Y 496.998,Z 416.619,A -85,B 0,C 180,E1 -6197.194,E2 -6197.194} C_VEL
LIN {X 0,Y 496.671,Z 427.297,A -85,B 0,C 180,E1 -6197.953,E2 -6197.953} C_VEL
LIN {X 0,Y 496.266,Z 437.762,A -85,B 0,C 180,E1 -6198.875,E2 -6198.875} C_VEL
LIN {X 0,Y 495.918,Z 446.314,A -85,B 0,C 180,E1 -6199.797,E2 -6199.797} C_VEL
LIN {X 0,Y 495.612,Z 454.201,A -85,B 0,C 180,E1 -6200.821,E2 -6200.821} C_VEL
LIN {X 0,Y 495.372,Z 461.898,A -85,B 0,C 180,E1 -6202.049,E2 -6202.049} C_VEL
LIN {X 0,Y 495.17,Z 468.986,A -85,B 0,C 180,E1 -6203.481,E2 -6203.481} C_VEL
LIN {X 0,Y 495.115,Z 473.702,A -85,B 0,C 180,E1 -6204.706,E2 -6204.706} C_VEL
LIN {X 0,Y 495.034,Z 477.303,A -85,B 0,C 180,E1 -6205.93,E2 -6205.93} C_VEL
LIN {X 0,Y 495.044,Z 479.161,A -85,B 0,C 180,E1 -6206.745,E2 -6206.745} C_VEL
LIN {X 0,Y 494.963,Z 481.545,A -85,B 0,C 180,E1 -6208.373,E2 -6208.373} C_VEL
LIN {X 0,Y 494.9,Z 482.365,A -85,B 0,C 180,E1 -6210,E2 -6210} C_VEL
LIN {X 0,Y 494.963,Z 481.542,A -85,B 0,C 180,E1 -6211.628,E2 -6211.628} C_VEL
LIN {X 0,Y 495.044,Z 479.154,A -85,B 0,C 180,E1 -6213.256,E2 -6213.256} C_VEL
LIN {X 0,Y 495.01,Z 476.222,A -85,B 0,C 180,E1 -6214.479,E2 -6214.479} C_VEL
LIN {X 0,Y 495.148,Z 472.254,A -85,B 0,C 180,E1 -6215.702,E2 -6215.702} C_VEL
LIN {X 0,Y 495.245,Z 466.147,A -85,B 0,C 180,E1 -6217.133,E2 -6217.133} C_VEL
LIN {X 0,Y 495.454,Z 459.478,A -85,B 0,C 180,E1 -6218.36,E2 -6218.36} C_VEL
LIN {X 0,Y 495.728,Z 451.204,A -85,B 0,C 180,E1 -6219.589,E2 -6219.589} C_VEL
LIN {X 0,Y 496.005,Z 442.718,A -85,B 0,C 180,E1 -6220.615,E2 -6220.615} C_VEL
LIN {X 0,Y 496.482,Z 432.233,A -85,B 0,C 180,E1 -6221.638,E2 -6221.638} C_VEL
LIN {X 0,Y 496.784,Z 420.804,A -85,B 0,C 180,E1 -6222.536,E2 -6222.536} C_VEL
LIN {X 0,Y 497.232,Z 408.547,A -85,B 0,C 180,E1 -6223.279,E2 -6223.279} C_VEL
LIN {X 0,Y 497.573,Z 396.186,A -85,B 0,C 180,E1 -6223.842,E2 -6223.842} C_VEL
LIN {X 0,Y 497.923,Z 383.482,A -85,B 0,C 180,E1 -6224.248,E2 -6224.248} C_VEL
LIN {X 0,Y 498.085,Z 370.143,A -85,B 0,C 180,E1 -6224.505,E2 -6224.505} C_VEL
LIN {X 0,Y 498.516,Z 284.101,A -85,B 0,C 180,E1 -6225.76,E2 -6225.76} C_VEL
LIN {X 0,Y 496.349,Z 270.717,A -85,B 0,C 180,E1 -6226.049,E2 -6226.049} C_VEL
LIN {X 0,Y 496.305,Z 269.622,A -85,B 0,C 180,E1 -6226.167,E2 -6226.167} C_VEL
LIN {X 0,Y 496.806,Z 252.132,A -85,B 0,C 180,E1 -6229.202,E2 -6229.202} C_VEL
LIN {X 0,Y 497.438,Z 235.137,A -85,B 0,C 180,E1 -6232.206,E2 -6232.206} C_VEL
LIN {X 0,Y 495.854,Z 225.533,A -85,B 0,C 180,E1 -6234.047,E2 -6234.047} C_VEL
LIN {X 0,Y 495.788,Z 225.23,A -85,B 0,C 180,E1 -6234.273,E2 -6234.273} C_VEL
LIN {X 0,Y 495.792,Z 225.227,A -85,B 0,C 180,E1 -6236.976,E2 -6236.976} C_VEL
LIN {X 0,Y 495.775,Z 225.231,A -85,B 0,C 180,E1 -6239.746,E2 -6239.746} C_VEL
LIN {X 0,Y 495.777,Z 225.224,A -85,B 0,C 180,E1 -6242.594,E2 -6242.594} C_VEL
LIN {X 0,Y 495.754,Z 225.229,A -85,B 0,C 180,E1 -6245.537,E2 -6245.537} C_VEL
LIN {X 0,Y 495.767,Z 225.225,A -85,B 0,C 180,E1 -6248.766,E2 -6248.766} C_VEL
LIN {X 0,Y 495.755,Z 225.229,A -85,B 0,C 180,E1 -6251.781,E2 -6251.781} C_VEL
LIN {X 0,Y 495.748,Z 225.229,A -85,B 0,C 180,E1 -6255.14,E2 -6255.14} C_VEL
LIN {X 0,Y 495.76,Z 225.223,A -85,B 0,C 180,E1 -6258.217,E2 -6258.217} C_VEL
LIN {X 0,Y 495.757,Z 225.225,A -85,B 0,C 180,E1 -6261.406,E2 -6261.406} C_VEL
LIN {X 0,Y 495.753,Z 225.231,A -85,B 0,C 180,E1 -6264.46,E2 -6264.46} C_VEL
LIN {X 0,Y 495.761,Z 225.226,A -85,B 0,C 180,E1 -6267.403,E2 -6267.403} C_VEL
LIN {X 0,Y 495.767,Z 225.226,A -85,B 0,C 180,E1 -6270.251,E2 -6270.251} C_VEL
LIN {X 0,Y 495.749,Z 225.234,A -85,B 0,C 180,E1 -6273.268,E2 -6273.268} C_VEL
LIN {X 0,Y 495.747,Z 225.226,A -85,B 0,C 180,E1 -6276.61,E2 -6276.61} C_VEL
LIN {X 0,Y 495.787,Z 225.227,A -85,B 0,C 180,E1 -6279.322,E2 -6279.322} C_VEL
LIN {X 0,Y 495.789,Z 225.226,A -85,B 0,C 180,E1 -6281.826,E2 -6281.826} C_VEL
LIN {X 0,Y 495.831,Z 225.213,A -85,B 0,C 180,E1 -6284.546,E2 -6284.546} C_VEL
LIN {X 0,Y 495.835,Z 225.218,A -85,B 0,C 180,E1 -6287.962,E2 -6287.962} C_VEL
LIN {X 0,Y 495.812,Z 225.22,A -85,B 0,C 180,E1 -6291.026,E2 -6291.026} C_VEL
LIN {X 0,Y 495.849,Z 225.218,A -85,B 0,C 180,E1 -6293.486,E2 -6293.486} C_VEL
LIN {X 0,Y 495.718,Z 225.24,A -85,B 0,C 180,E1 -6295.932,E2 -6295.932} C_VEL
LIN {X 0,Y 495.986,Z 225.201,A -85,B 0,C 180,E1 -6297.56,E2 -6297.56} C_VEL
LIN {X 0,Y 495.941,Z 225.204,A -85,B 0,C 180,E1 -6300.808,E2 -6300.808} C_VEL
LIN {X 0,Y 495.985,Z 225.199,A -85,B 0,C 180,E1 -6302.433,E2 -6302.433} C_VEL
LIN {X 0,Y 495.878,Z 225.213,A -85,B 0,C 180,E1 -6305.69,E2 -6305.69} C_VEL
LIN {X 0,Y 495.832,Z 225.219,A -85,B 0,C 180,E1 -6308.966,E2 -6308.966} C_VEL
LIN {X 0,Y 495.822,Z 225.218,A -85,B 0,C 180,E1 -6312.031,E2 -6312.031} C_VEL
LIN {X 0,Y 495.815,Z 225.217,A -85,B 0,C 180,E1 -6315.447,E2 -6315.447} C_VEL
LIN {X 0,Y 495.767,Z 225.228,A -85,B 0,C 180,E1 -6318.233,E2 -6318.233} C_VEL
LIN {X 0,Y 495.762,Z 225.235,A -85,B 0,C 180,E1 -6320.752,E2 -6320.752} C_VEL
LIN {X 0,Y 495.74,Z 225.231,A -85,B 0,C 180,E1 -6323.383,E2 -6323.383} C_VEL
LIN {X 0,Y 495.773,Z 225.217,A -85,B 0,C 180,E1 -6326.063,E2 -6326.063} C_VEL
LIN {X 0,Y 495.753,Z 225.232,A -85,B 0,C 180,E1 -6328.81,E2 -6328.81} C_VEL
LIN {X 0,Y 495.734,Z 225.231,A -85,B 0,C 180,E1 -6331.721,E2 -6331.721} C_VEL
LIN {X 0,Y 495.751,Z 225.228,A -85,B 0,C 180,E1 -6334.691,E2 -6334.691} C_VEL
LIN {X 0,Y 495.708,Z 225.236,A -85,B 0,C 180,E1 -6337.557,E2 -6337.557} C_VEL
LIN {X 0,Y 495.773,Z 225.226,A -85,B 0,C 180,E1 -6340.049,E2 -6340.049} C_VEL
LIN {X 0,Y 495.733,Z 225.232,A -85,B 0,C 180,E1 -6342.875,E2 -6342.875} C_VEL
LIN {X 0,Y 495.703,Z 225.239,A -85,B 0,C 180,E1 -6345.995,E2 -6345.995} C_VEL
LIN {X 0,Y 495.739,Z 225.233,A -85,B 0,C 180,E1 -6348.701,E2 -6348.701} C_VEL
LIN {X 0,Y 495.828,Z 225.415,A -85,B 0,C 180,E1 -6350.008,E2 -6350.008} C_VEL
LIN {X 0,Y 496.882,Z 231.944,A -85,B 0,C 180,E1 -6351.299,E2 -6351.299} C_VEL
LIN {X 0,Y 496.584,Z 246.674,A -85,B 0,C 180,E1 -6354.034,E2 -6354.034} C_VEL
LIN {X 0,Y 496.286,Z 257.488,A -85,B 0,C 180,E1 -6355.967,E2 -6355.967} C_VEL
LIN {X 0,Y 497.063,Z 261.872,A -85,B 0,C 180,E1 -6356.099,E2 -6356.099} C_VEL
LIN {X 0,Y 498.592,Z 270.558,A -85,B 0,C 180,E1 -6356.282,E2 -6356.282} C_VEL
LIN {X 0,Y 498.518,Z 287.706,A -85,B 0,C 180,E1 -6356.535,E2 -6356.535} C_VEL
LIN {X 0,Y 497.871,Z 293.55,A -85,B 0,C 180,E1 -6356.6,E2 -6356.6} C_VEL
LIN {X 0,Y 492.224,Z 312.556,A -85,B 0,C 180,E1 -6356.696,E2 -6356.696} C_VEL
LIN {X 0,Y 491.516,Z 318.402,A -85,B 0,C 180,E1 -6356.761,E2 -6356.761} C_VEL
LIN {X 0,Y 491.11,Z 365.864,A -85,B 0,C 180,E1 -6357.486,E2 -6357.486} C_VEL
LIN {X 0,Y 490.862,Z 379.482,A -85,B 0,C 180,E1 -6357.874,E2 -6357.874} C_VEL
LIN {X 0,Y 490.521,Z 392.092,A -85,B 0,C 180,E1 -6358.409,E2 -6358.409} C_VEL
LIN {X 0,Y 490.109,Z 404.54,A -85,B 0,C 180,E1 -6359.13,E2 -6359.13} C_VEL
LIN {X 0,Y 489.703,Z 415.783,A -85,B 0,C 180,E1 -6359.966,E2 -6359.966} C_VEL
LIN {X 0,Y 489.274,Z 425.788,A -85,B 0,C 180,E1 -6360.896,E2 -6360.896} C_VEL
LIN {X 0,Y 488.939,Z 434.717,A -85,B 0,C 180,E1 -6361.917,E2 -6361.917} C_VEL
LIN {X 0,Y 488.557,Z 443.165,A -85,B 0,C 180,E1 -6363.097,E2 -6363.097} C_VEL
LIN {X 0,Y 488.299,Z 450.775,A -85,B 0,C 180,E1 -6364.419,E2 -6364.419} C_VEL
LIN {X 0,Y 488.125,Z 456.871,A -85,B 0,C 180,E1 -6365.774,E2 -6365.774} C_VEL
LIN {X 0,Y 487.975,Z 461.692,A -85,B 0,C 180,E1 -6367.168,E2 -6367.168} C_VEL
LIN {X 0,Y 487.922,Z 463.966,A -85,B 0,C 180,E1 -6368.006,E2 -6368.006} C_VEL
LIN {X 0,Y 487.882,Z 466.764,A -85,B 0,C 180,E1 -6369.427,E2 -6369.427} C_VEL
LIN {X 0,Y 487.81,Z 468.187,A -85,B 0,C 180,E1 -6370.648,E2 -6370.648} C_VEL
LIN {X 0,Y 487.79,Z 468.742,A -85,B 0,C 180,E1 -6371.954,E2 -6371.954} C_VEL
LIN {X 0,Y 487.79,Z 468.313,A -85,B 0,C 180,E1 -6373.252,E2 -6373.252} C_VEL
LIN {X 0,Y 487.897,Z 466.524,A -85,B 0,C 180,E1 -6374.797,E2 -6374.797} C_VEL
LIN {X 0,Y 487.95,Z 463.502,A -85,B 0,C 180,E1 -6376.252,E2 -6376.252} C_VEL
LIN {X 0,Y 488.008,Z 459.741,A -85,B 0,C 180,E1 -6377.524,E2 -6377.524} C_VEL
LIN {X 0,Y 488.19,Z 454.826,A -85,B 0,C 180,E1 -6378.793,E2 -6378.793} C_VEL
LIN {X 0,Y 488.369,Z 448.645,A -85,B 0,C 180,E1 -6380.056,E2 -6380.056} C_VEL
LIN {X 0,Y 488.68,Z 440.958,A -85,B 0,C 180,E1 -6381.314,E2 -6381.314} C_VEL
LIN {X 0,Y 489.074,Z 431.306,A -85,B 0,C 180,E1 -6382.569,E2 -6382.569} C_VEL
LIN {X 0,Y 489.42,Z 421.392,A -85,B 0,C 180,E1 -6383.61,E2 -6383.61} C_VEL
LIN {X 0,Y 489.878,Z 410.198,A -85,B 0,C 180,E1 -6384.546,E2 -6384.546} C_VEL
LIN {X 0,Y 490.281,Z 399.249,A -85,B 0,C 180,E1 -6385.272,E2 -6385.272} C_VEL
LIN {X 0,Y 490.659,Z 387.153,A -85,B 0,C 180,E1 -6385.893,E2 -6385.893} C_VEL
LIN {X 0,Y 490.912,Z 374.668,A -85,B 0,C 180,E1 -6386.357,E2 -6386.357} C_VEL
LIN {X 0,Y 491.176,Z 361.474,A -85,B 0,C 180,E1 -6386.667,E2 -6386.667} C_VEL
LIN {X 0,Y 491.652,Z 270.835,A -85,B 0,C 180,E1 -6388.003,E2 -6388.003} C_VEL
LIN {X 0,Y 489.537,Z 259.199,A -85,B 0,C 180,E1 -6388.252,E2 -6388.252} C_VEL
LIN {X 0,Y 489.307,Z 257.425,A -85,B 0,C 180,E1 -6388.354,E2 -6388.354} C_VEL
LIN {X 0,Y 489.752,Z 242.324,A -85,B 0,C 180,E1 -6391.233,E2 -6391.233} C_VEL
LIN {X 0,Y 490.002,Z 232.778,A -85,B 0,C 180,E1 -6393.083,E2 -6393.083} C_VEL
LIN {X 0,Y 488.791,Z 226.189,A -85,B 0,C 180,E1 -6394.484,E2 -6394.484} C_VEL
LIN {X 0,Y 488.841,Z 226.095,A -85,B 0,C 180,E1 -6396.604,E2 -6396.604} C_VEL
LIN {X 0,Y 488.772,Z 226.1,A -85,B 0,C 180,E1 -6399.1,E2 -6399.1} C_VEL
LIN {X 0,Y 488.768,Z 226.103,A -85,B 0,C 180,E1 -6402.455,E2 -6402.455} C_VEL
LIN {X 0,Y 488.748,Z 226.1,A -85,B 0,C 180,E1 -6405.566,E2 -6405.566} C_VEL
LIN {X 0,Y 488.719,Z 226.104,A -85,B 0,C 180,E1 -6408.443,E2 -6408.443} C_VEL
LIN {X 0,Y 488.72,Z 226.109,A -85,B 0,C 180,E1 -6411.07,E2 -6411.07} C_VEL
LIN {X 0,Y 488.677,Z 226.107,A -85,B 0,C 180,E1 -6413.746,E2 -6413.746} C_VEL
LIN {X 0,Y 488.754,Z 226.09,A -85,B 0,C 180,E1 -6416.948,E2 -6416.948} C_VEL
LIN {X 0,Y 488.709,Z 226.103,A -85,B 0,C 180,E1 -6420.22,E2 -6420.22} C_VEL
LIN {X 0,Y 488.713,Z 226.11,A -85,B 0,C 180,E1 -6423.491,E2 -6423.491} C_VEL
LIN {X 0,Y 488.668,Z 226.107,A -85,B 0,C 180,E1 -6426.362,E2 -6426.362} C_VEL
LIN {X 0,Y 488.721,Z 226.106,A -85,B 0,C 180,E1 -6429.252,E2 -6429.252} C_VEL
LIN {X 0,Y 488.708,Z 226.097,A -85,B 0,C 180,E1 -6432.523,E2 -6432.523} C_VEL
LIN {X 0,Y 488.695,Z 226.105,A -85,B 0,C 180,E1 -6435.204,E2 -6435.204} C_VEL
LIN {X 0,Y 488.712,Z 226.106,A -85,B 0,C 180,E1 -6437.484,E2 -6437.484} C_VEL
LIN {X 0,Y 488.719,Z 226.093,A -85,B 0,C 180,E1 -6440.754,E2 -6440.754} C_VEL
LIN {X 0,Y 488.663,Z 226.108,A -85,B 0,C 180,E1 -6443.873,E2 -6443.873} C_VEL
LIN {X 0,Y 488.714,Z 226.105,A -85,B 0,C 180,E1 -6446.881,E2 -6446.881} C_VEL
LIN {X 0,Y 488.71,Z 226.101,A -85,B 0,C 180,E1 -6449.786,E2 -6449.786} C_VEL
LIN {X 0,Y 488.777,Z 226.089,A -85,B 0,C 180,E1 -6453.059,E2 -6453.059} C_VEL
LIN {X 0,Y 488.682,Z 226.107,A -85,B 0,C 180,E1 -6456.259,E2 -6456.259} C_VEL
LIN {X 0,Y 488.731,Z 226.105,A -85,B 0,C 180,E1 -6459.179,E2 -6459.179} C_VEL
LIN {X 0,Y 488.744,Z 226.095,A -85,B 0,C 180,E1 -6461.632,E2 -6461.632} C_VEL
LIN {X 0,Y 488.749,Z 226.09,A -85,B 0,C 180,E1 -6465.004,E2 -6465.004} C_VEL
LIN {X 0,Y 488.821,Z 226.086,A -85,B 0,C 180,E1 -6468.392,E2 -6468.392} C_VEL
LIN {X 0,Y 488.811,Z 226.094,A -85,B 0,C 180,E1 -6471.738,E2 -6471.738} C_VEL
LIN {X 0,Y 488.852,Z 226.082,A -85,B 0,C 180,E1 -6474.228,E2 -6474.228} C_VEL
LIN {X 0,Y 488.956,Z 226.065,A -85,B 0,C 180,E1 -6477.532,E2 -6477.532} C_VEL
LIN {X 0,Y 488.931,Z 226.071,A -85,B 0,C 180,E1 -6480.827,E2 -6480.827} C_VEL
LIN {X 0,Y 488.959,Z 226.073,A -85,B 0,C 180,E1 -6482.475,E2 -6482.475} C_VEL
LIN {X 0,Y 488.84,Z 226.095,A -85,B 0,C 180,E1 -6485.779,E2 -6485.779} C_VEL
LIN {X 0,Y 488.816,Z 226.086,A -85,B 0,C 180,E1 -6488.27,E2 -6488.27} C_VEL
LIN {X 0,Y 488.807,Z 226.083,A -85,B 0,C 180,E1 -6491.616,E2 -6491.616} C_VEL
LIN {X 0,Y 488.765,Z 226.097,A -85,B 0,C 180,E1 -6495.003,E2 -6495.003} C_VEL
LIN {X 0,Y 488.751,Z 226.102,A -85,B 0,C 180,E1 -6498.445,E2 -6498.445} C_VEL
LIN {X 0,Y 488.712,Z 226.097,A -85,B 0,C 180,E1 -6501.073,E2 -6501.073} C_VEL
LIN {X 0,Y 488.688,Z 226.105,A -85,B 0,C 180,E1 -6503.749,E2 -6503.749} C_VEL
LIN {X 0,Y 488.752,Z 226.104,A -85,B 0,C 180,E1 -6506.935,E2 -6506.935} C_VEL
LIN {X 0,Y 488.728,Z 226.097,A -85,B 0,C 180,E1 -6509.273,E2 -6509.273} C_VEL
LIN {X 0,Y 488.703,Z 226.104,A -85,B 0,C 180,E1 -6512.15,E2 -6512.15} C_VEL
LIN {X 0,Y 488.72,Z 226.11,A -85,B 0,C 180,E1 -6515.117,E2 -6515.117} C_VEL
LIN {X 0,Y 488.683,Z 226.105,A -85,B 0,C 180,E1 -6518.202,E2 -6518.202} C_VEL
LIN {X 0,Y 488.726,Z 226.102,A -85,B 0,C 180,E1 -6520.346,E2 -6520.346} C_VEL
LIN {X 0,Y 488.685,Z 226.1,A -85,B 0,C 180,E1 -6523.657,E2 -6523.657} C_VEL
LIN {X 0,Y 488.684,Z 226.1,A -85,B 0,C 180,E1 -6526.346,E2 -6526.346} C_VEL
LIN {X 0,Y 488.711,Z 226.112,A -85,B 0,C 180,E1 -6529.675,E2 -6529.675} C_VEL
LIN {X 0,Y 488.677,Z 226.107,A -85,B 0,C 180,E1 -6532.841,E2 -6532.841} C_VEL
LIN {X 0,Y 488.737,Z 226.106,A -85,B 0,C 180,E1 -6535.888,E2 -6535.888} C_VEL
LIN {X 0,Y 488.698,Z 226.107,A -85,B 0,C 180,E1 -6538.821,E2 -6538.821} C_VEL
LIN {X 0,Y 488.749,Z 226.105,A -85,B 0,C 180,E1 -6541.672,E2 -6541.672} C_VEL
LIN {X 0,Y 488.716,Z 226.112,A -85,B 0,C 180,E1 -6544.443,E2 -6544.443} C_VEL
LIN {X 0,Y 488.749,Z 226.15,A -85,B 0,C 180,E1 -6545.694,E2 -6545.694} C_VEL
LIN {X 0,Y 489.271,Z 228.897,A -85,B 0,C 180,E1 -6546.285,E2 -6546.285} C_VEL
LIN {X 0,Y 490.456,Z 236.236,A -85,B 0,C 180,E1 -6547.683,E2 -6547.683} C_VEL
LIN {X 0,Y 489.759,Z 256.343,A -85,B 0,C 180,E1 -6551.283,E2 -6551.283} C_VEL
LIN {X 0,Y 489.335,Z 270.47,A -85,B 0,C 180,E1 -6553.736,E2 -6553.736} C_VEL
LIN {X 0,Y 491.676,Z 286.109,A -85,B 0,C 180,E1 -6554.066,E2 -6554.066} C_VEL
LIN {X 0,Y 491.115,Z 378.373,A -85,B 0,C 180,E1 -6555.444,E2 -6555.444} C_VEL
LIN {X 0,Y 490.817,Z 391.54,A -85,B 0,C 180,E1 -6555.806,E2 -6555.806} C_VEL
LIN {X 0,Y 490.454,Z 404.217,A -85,B 0,C 180,E1 -6556.324,E2 -6556.324} C_VEL
LIN {X 0,Y 490.09,Z 415.636,A -85,B 0,C 180,E1 -6556.957,E2 -6556.957} C_VEL
LIN {X 0,Y 489.699,Z 427.133,A -85,B 0,C 180,E1 -6557.779,E2 -6557.779} C_VEL
LIN {X 0,Y 489.285,Z 437.61,A -85,B 0,C 180,E1 -6558.714,E2 -6558.714} C_VEL
LIN {X 0,Y 488.885,Z 446.171,A -85,B 0,C 180,E1 -6559.648,E2 -6559.648} C_VEL
LIN {X 0,Y 488.565,Z 454.067,A -85,B 0,C 180,E1 -6560.687,E2 -6560.687} C_VEL
LIN {X 0,Y 488.325,Z 461.776,A -85,B 0,C 180,E1 -6561.934,E2 -6561.934} C_VEL
LIN {X 0,Y 488.103,Z 468.872,A -85,B 0,C 180,E1 -6563.386,E2 -6563.386} C_VEL
LIN {X 0,Y 488.049,Z 473.594,A -85,B 0,C 180,E1 -6564.629,E2 -6564.629} C_VEL
LIN {X 0,Y 487.93,Z 477.198,A -85,B 0,C 180,E1 -6565.87,E2 -6565.87} C_VEL
LIN {X 0,Y 487.967,Z 479.059,A -85,B 0,C 180,E1 -6566.698,E2 -6566.698} C_VEL
LIN {X 0,Y 487.891,Z 481.446,A -85,B 0,C 180,E1 -6568.349,E2 -6568.349} C_VEL
LIN {X 0,Y 487.821,Z 482.267,A -85,B 0,C 180,E1 -6570,E2 -6570} C_VEL
LIN {X 0,Y 487.891,Z 481.445,A -85,B 0,C 180,E1 -6571.651,E2 -6571.651} C_VEL
LIN {X 0,Y 487.967,Z 479.059,A -85,B 0,C 180,E1 -6573.303,E2 -6573.303} C_VEL
LIN {X 0,Y 487.923,Z 476.128,A -85,B 0,C 180,E1 -6574.544,E2 -6574.544} C_VEL
LIN {X 0,Y 488.065,Z 472.162,A -85,B 0,C 180,E1 -6575.785,E2 -6575.785} C_VEL
LIN {X 0,Y 488.134,Z 467.058,A -85,B 0,C 180,E1 -6577.03,E2 -6577.03} C_VEL
LIN {X 0,Y 488.346,Z 460.63,A -85,B 0,C 180,E1 -6578.275,E2 -6578.275} C_VEL
LIN {X 0,Y 488.623,Z 452.612,A -85,B 0,C 180,E1 -6579.521,E2 -6579.521} C_VEL
LIN {X 0,Y 488.943,Z 444.44,A -85,B 0,C 180,E1 -6580.56,E2 -6580.56} C_VEL
LIN {X 0,Y 489.381,Z 434.476,A -85,B 0,C 180,E1 -6581.599,E2 -6581.599} C_VEL
LIN {X 0,Y 489.755,Z 424.642,A -85,B 0,C 180,E1 -6582.43,E2 -6582.43} C_VEL
LIN {X 0,Y 490.148,Z 414.121,A -85,B 0,C 180,E1 -6583.148,E2 -6583.148} C_VEL
LIN {X 0,Y 490.511,Z 402.229,A -85,B 0,C 180,E1 -6583.781,E2 -6583.781} C_VEL
LIN {X 0,Y 490.918,Z 388.895,A -85,B 0,C 180,E1 -6584.297,E2 -6584.297} C_VEL
LIN {X 0,Y 491.162,Z 376.526,A -85,B 0,C 180,E1 -6584.608,E2 -6584.608} C_VEL
LIN {X 0,Y 491.739,Z 284.971,A -85,B 0,C 180,E1 -6585.975,E2 -6585.975} C_VEL
LIN {X 0,Y 489.346,Z 270.389,A -85,B 0,C 180,E1 -6586.307,E2 -6586.307} C_VEL
LIN {X 0,Y 489.51,Z 263.006,A -85,B 0,C 180,E1 -6587.548,E2 -6587.548} C_VEL
LIN {X 0,Y 490.133,Z 244.811,A -85,B 0,C 180,E1 -6590.787,E2 -6590.787} C_VEL
LIN {X 0,Y 490.503,Z 236.335,A -85,B 0,C 180,E1 -6592.315,E2 -6592.315} C_VEL
LIN {X 0,Y 488.783,Z 226.244,A -85,B 0,C 180,E1 -6594.305,E2 -6594.305} C_VEL
LIN {X 0,Y 488.74,Z 226.107,A -85,B 0,C 180,E1 -6597.397,E2 -6597.397} C_VEL
LIN {X 0,Y 488.717,Z 226.106,A -85,B 0,C 180,E1 -6600.361,E2 -6600.361} C_VEL
LIN {X 0,Y 488.745,Z 226.1,A -85,B 0,C 180,E1 -6603.483,E2 -6603.483} C_VEL
LIN {X 0,Y 488.683,Z 226.115,A -85,B 0,C 180,E1 -6606.352,E2 -6606.352} C_VEL
LIN {X 0,Y 488.704,Z 226.103,A -85,B 0,C 180,E1 -6609.254,E2 -6609.254} C_VEL
LIN {X 0,Y 488.698,Z 226.107,A -85,B 0,C 180,E1 -6612.525,E2 -6612.525} C_VEL
LIN {X 0,Y 488.712,Z 226.105,A -85,B 0,C 180,E1 -6615.196,E2 -6615.196} C_VEL
LIN {X 0,Y 488.703,Z 226.107,A -85,B 0,C 180,E1 -6618.581,E2 -6618.581} C_VEL
LIN {X 0,Y 488.711,Z 226.107,A -85,B 0,C 180,E1 -6620.947,E2 -6620.947} C_VEL
LIN {X 0,Y 488.679,Z 226.108,A -85,B 0,C 180,E1 -6623.865,E2 -6623.865} C_VEL
LIN {X 0,Y 488.712,Z 226.111,A -85,B 0,C 180,E1 -6626.873,E2 -6626.873} C_VEL
LIN {X 0,Y 488.728,Z 226.103,A -85,B 0,C 180,E1 -6629.778,E2 -6629.778} C_VEL
LIN {X 0,Y 488.707,Z 226.111,A -85,B 0,C 180,E1 -6633.076,E2 -6633.076} C_VEL
LIN {X 0,Y 488.677,Z 226.105,A -85,B 0,C 180,E1 -6636.251,E2 -6636.251} C_VEL
LIN {X 0,Y 488.755,Z 226.105,A -85,B 0,C 180,E1 -6639.173,E2 -6639.173} C_VEL
LIN {X 0,Y 488.757,Z 226.104,A -85,B 0,C 180,E1 -6641.629,E2 -6641.629} C_VEL
LIN {X 0,Y 488.767,Z 226.095,A -85,B 0,C 180,E1 -6644.997,E2 -6644.997} C_VEL
LIN {X 0,Y 488.811,Z 226.089,A -85,B 0,C 180,E1 -6648.384,E2 -6648.384} C_VEL
LIN {X 0,Y 488.779,Z 226.104,A -85,B 0,C 180,E1 -6651.73,E2 -6651.73} C_VEL
LIN {X 0,Y 488.839,Z 226.09,A -85,B 0,C 180,E1 -6654.221,E2 -6654.221} C_VEL
LIN {X 0,Y 488.953,Z 226.077,A -85,B 0,C 180,E1 -6657.525,E2 -6657.525} C_VEL
LIN {X 0,Y 488.97,Z 226.078,A -85,B 0,C 180,E1 -6659.996,E2 -6659.996} C_VEL
LIN {X 0,Y 488.952,Z 226.074,A -85,B 0,C 180,E1 -6662.468,E2 -6662.468} C_VEL
LIN {X 0,Y 488.835,Z 226.091,A -85,B 0,C 180,E1 -6665.772,E2 -6665.772} C_VEL
LIN {X 0,Y 488.781,Z 226.099,A -85,B 0,C 180,E1 -6668.263,E2 -6668.263} C_VEL
LIN {X 0,Y 488.799,Z 226.089,A -85,B 0,C 180,E1 -6671.608,E2 -6671.608} C_VEL
LIN {X 0,Y 488.756,Z 226.1,A -85,B 0,C 180,E1 -6674.996,E2 -6674.996} C_VEL
LIN {X 0,Y 488.735,Z 226.106,A -85,B 0,C 180,E1 -6678.438,E2 -6678.438} C_VEL
LIN {X 0,Y 488.696,Z 226.109,A -85,B 0,C 180,E1 -6681.066,E2 -6681.066} C_VEL
LIN {X 0,Y 488.679,Z 226.109,A -85,B 0,C 180,E1 -6683.741,E2 -6683.741} C_VEL
LIN {X 0,Y 488.774,Z 226.095,A -85,B 0,C 180,E1 -6686.939,E2 -6686.939} C_VEL
LIN {X 0,Y 488.688,Z 226.106,A -85,B 0,C 180,E1 -6690.358,E2 -6690.358} C_VEL
LIN {X 0,Y 488.712,Z 226.109,A -85,B 0,C 180,E1 -6693.48,E2 -6693.48} C_VEL
LIN {X 0,Y 488.663,Z 226.111,A -85,B 0,C 180,E1 -6696.351,E2 -6696.351} C_VEL
LIN {X 0,Y 488.723,Z 226.107,A -85,B 0,C 180,E1 -6699.245,E2 -6699.245} C_VEL
LIN {X 0,Y 488.703,Z 226.112,A -85,B 0,C 180,E1 -6701.599,E2 -6701.599} C_VEL
LIN {X 0,Y 488.67,Z 226.115,A -85,B 0,C 180,E1 -6704.02,E2 -6704.02} C_VEL
LIN {X 0,Y 488.711,Z 226.109,A -85,B 0,C 180,E1 -6707.165,E2 -6707.165} C_VEL
LIN {X 0,Y 488.769,Z 226.168,A -85,B 0,C 180,E1 -6709.766,E2 -6709.766} C_VEL
LIN {X 0,Y 489.706,Z 231.289,A -85,B 0,C 180,E1 -6710.842,E2 -6710.842} C_VEL
LIN {X 0,Y 489.905,Z 236.897,A -85,B 0,C 180,E1 -6711.913,E2 -6711.913} C_VEL
LIN {X 0,Y 489.425,Z 253.112,A -85,B 0,C 180,E1 -6714.943,E2 -6714.943} C_VEL
LIN {X 0,Y 489.351,Z 257.582,A -85,B 0,C 180,E1 -6715.726,E2 -6715.726} C_VEL
LIN {X 0,Y 490.184,Z 262.238,A -85,B 0,C 180,E1 -6715.866,E2 -6715.866} C_VEL
LIN {X 0,Y 491.787,Z 272.332,A -85,B 0,C 180,E1 -6716.077,E2 -6716.077} C_VEL
LIN {X 0,Y 491.516,Z 318.402,A -85,B 0,C 180,E1 -6716.761,E2 -6716.761} C_VEL
LIN {X 0,Y 490.807,Z 324.247,A -85,B 0,C 180,E1 -6716.824,E2 -6716.824} C_VEL
LIN {X 0,Y 485.115,Z 343.242,A -85,B 0,C 180,E1 -6716.92,E2 -6716.92} C_VEL
LIN {X 0,Y 484.434,Z 349.085,A -85,B 0,C 180,E1 -6716.986,E2 -6716.986} C_VEL
LIN {X 0,Y 484.258,Z 368.057,A -85,B 0,C 180,E1 -6717.314,E2 -6717.314} C_VEL
LIN {X 0,Y 483.995,Z 380.387,A -85,B 0,C 180,E1 -6717.687,E2 -6717.687} C_VEL
LIN {X 0,Y 483.645,Z 392.419,A -85,B 0,C 180,E1 -6718.213,E2 -6718.213} C_VEL
LIN {X 0,Y 483.191,Z 404.511,A -85,B 0,C 180,E1 -6718.924,E2 -6718.924} C_VEL
LIN {X 0,Y 482.78,Z 415.271,A -85,B 0,C 180,E1 -6719.732,E2 -6719.732} C_VEL
LIN {X 0,Y 482.335,Z 425.5,A -85,B 0,C 180,E1 -6720.685,E2 -6720.685} C_VEL
LIN {X 0,Y 481.956,Z 434.41,A -85,B 0,C 180,E1 -6721.711,E2 -6721.711} C_VEL
LIN {X 0,Y 481.544,Z 442.832,A -85,B 0,C 180,E1 -6722.895,E2 -6722.895} C_VEL
LIN {X 0,Y 481.247,Z 450.597,A -85,B 0,C 180,E1 -6724.249,E2 -6724.249} C_VEL
LIN {X 0,Y 481.069,Z 455.845,A -85,B 0,C 180,E1 -6725.395,E2 -6725.395} C_VEL
LIN {X 0,Y 480.923,Z 460.812,A -85,B 0,C 180,E1 -6726.761,E2 -6726.761} C_VEL
LIN {X 0,Y 480.827,Z 464.467,A -85,B 0,C 180,E1 -6728.116,E2 -6728.116} C_VEL
LIN {X 0,Y 480.791,Z 466.968,A -85,B 0,C 180,E1 -6729.462,E2 -6729.462} C_VEL
LIN {X 0,Y 480.72,Z 468.026,A -85,B 0,C 180,E1 -6730.351,E2 -6730.351} C_VEL
LIN {X 0,Y 480.704,Z 468.821,A -85,B 0,C 180,E1 -6731.843,E2 -6731.843} C_VEL
LIN {X 0,Y 480.691,Z 468.565,A -85,B 0,C 180,E1 -6732.997,E2 -6732.997} C_VEL
LIN {X 0,Y 480.724,Z 467.878,A -85,B 0,C 180,E1 -6733.872,E2 -6733.872} C_VEL
LIN {X 0,Y 480.804,Z 466.77,A -85,B 0,C 180,E1 -6734.745,E2 -6734.745} C_VEL
LIN {X 0,Y 480.844,Z 464.262,A -85,B 0,C 180,E1 -6736.045,E2 -6736.045} C_VEL
LIN {X 0,Y 480.917,Z 460.722,A -85,B 0,C 180,E1 -6737.337,E2 -6737.337} C_VEL
LIN {X 0,Y 481.094,Z 456.049,A -85,B 0,C 180,E1 -6738.626,E2 -6738.626} C_VEL
LIN {X 0,Y 481.315,Z 448.994,A -85,B 0,C 180,E1 -6740.121,E2 -6740.121} C_VEL
LIN {X 0,Y 481.651,Z 441.366,A -85,B 0,C 180,E1 -6741.398,E2 -6741.398} C_VEL
LIN {X 0,Y 481.99,Z 433.367,A -85,B 0,C 180,E1 -6742.485,E2 -6742.485} C_VEL
LIN {X 0,Y 482.276,Z 424.127,A -85,B 0,C 180,E1 -6743.515,E2 -6743.515} C_VEL
LIN {X 0,Y 482.751,Z 413.586,A -85,B 0,C 180,E1 -6744.465,E2 -6744.465} C_VEL
LIN {X 0,Y 483.243,Z 401.85,A -85,B 0,C 180,E1 -6745.307,E2 -6745.307} C_VEL
LIN {X 0,Y 483.696,Z 389.297,A -85,B 0,C 180,E1 -6745.99,E2 -6745.99} C_VEL
LIN {X 0,Y 483.998,Z 376.851,A -85,B 0,C 180,E1 -6746.488,E2 -6746.488} C_VEL
LIN {X 0,Y 484.241,Z 364.013,A -85,B 0,C 180,E1 -6746.828,E2 -6746.828} C_VEL
LIN {X 0,Y 484.847,Z 271.961,A -85,B 0,C 180,E1 -6748.209,E2 -6748.209} C_VEL
LIN {X 0,Y 482.399,Z 258.499,A -85,B 0,C 180,E1 -6748.513,E2 -6748.513} C_VEL
LIN {X 0,Y 482.322,Z 257.167,A -85,B 0,C 180,E1 -6748.643,E2 -6748.643} C_VEL
LIN {X 0,Y 482.862,Z 241.561,A -85,B 0,C 180,E1 -6751.668,E2 -6751.668} C_VEL
LIN {X 0,Y 483.04,Z 234.149,A -85,B 0,C 180,E1 -6753.127,E2 -6753.127} C_VEL
LIN {X 0,Y 481.782,Z 227.001,A -85,B 0,C 180,E1 -6754.68,E2 -6754.68} C_VEL
LIN {X 0,Y 481.793,Z 226.967,A -85,B 0,C 180,E1 -6757.544,E2 -6757.544} C_VEL
LIN {X 0,Y 481.706,Z 226.981,A -85,B 0,C 180,E1 -6760.933,E2 -6760.933} C_VEL
LIN {X 0,Y 481.697,Z 226.979,A -85,B 0,C 180,E1 -6763.499,E2 -6763.499} C_VEL
LIN {X 0,Y 481.675,Z 226.982,A -85,B 0,C 180,E1 -6766.094,E2 -6766.094} C_VEL
LIN {X 0,Y 481.67,Z 226.98,A -85,B 0,C 180,E1 -6768.723,E2 -6768.723} C_VEL
LIN {X 0,Y 481.655,Z 226.986,A -85,B 0,C 180,E1 -6771.394,E2 -6771.394} C_VEL
LIN {X 0,Y 481.656,Z 226.981,A -85,B 0,C 180,E1 -6774.114,E2 -6774.114} C_VEL
LIN {X 0,Y 481.707,Z 226.967,A -85,B 0,C 180,E1 -6777.143,E2 -6777.143} C_VEL
LIN {X 0,Y 481.66,Z 226.984,A -85,B 0,C 180,E1 -6779.742,E2 -6779.742} C_VEL
LIN {X 0,Y 481.657,Z 226.984,A -85,B 0,C 180,E1 -6782.675,E2 -6782.675} C_VEL
LIN {X 0,Y 481.621,Z 226.991,A -85,B 0,C 180,E1 -6785.71,E2 -6785.71} C_VEL
LIN {X 0,Y 481.679,Z 226.98,A -85,B 0,C 180,E1 -6788.858,E2 -6788.858} C_VEL
LIN {X 0,Y 481.645,Z 226.98,A -85,B 0,C 180,E1 -6792.16,E2 -6792.16} C_VEL
LIN {X 0,Y 481.663,Z 226.982,A -85,B 0,C 180,E1 -6794.456,E2 -6794.456} C_VEL
LIN {X 0,Y 481.702,Z 226.977,A -85,B 0,C 180,E1 -6796.843,E2 -6796.843} C_VEL
LIN {X 0,Y 481.681,Z 226.979,A -85,B 0,C 180,E1 -6800.067,E2 -6800.067} C_VEL
LIN {X 0,Y 481.608,Z 226.983,A -85,B 0,C 180,E1 -6803.379,E2 -6803.379} C_VEL
LIN {X 0,Y 481.682,Z 226.988,A -85,B 0,C 180,E1 -6806.334,E2 -6806.334} C_VEL
LIN {X 0,Y 481.634,Z 226.981,A -85,B 0,C 180,E1 -6809.42,E2 -6809.42} C_VEL
LIN {X 0,Y 481.681,Z 226.971,A -85,B 0,C 180,E1 -6812.173,E2 -6812.173} C_VEL
LIN {X 0,Y 481.7,Z 226.979,A -85,B 0,C 180,E1 -6814.974,E2 -6814.974} C_VEL
LIN {X 0,Y 481.642,Z 226.984,A -85,B 0,C 180,E1 -6817.71,E2 -6817.71} C_VEL
LIN {X 0,Y 481.693,Z 226.979,A -85,B 0,C 180,E1 -6820.397,E2 -6820.397} C_VEL
LIN {X 0,Y 481.679,Z 226.974,A -85,B 0,C 180,E1 -6823.038,E2 -6823.038} C_VEL
LIN {X 0,Y 481.677,Z 226.97,A -85,B 0,C 180,E1 -6825.643,E2 -6825.643} C_VEL
LIN {X 0,Y 481.785,Z 226.962,A -85,B 0,C 180,E1 -6828.22,E2 -6828.22} C_VEL
LIN {X 0,Y 481.756,Z 226.974,A -85,B 0,C 180,E1 -6831.616,E2 -6831.616} C_VEL
LIN {X 0,Y 481.813,Z 226.959,A -85,B 0,C 180,E1 -6834.144,E2 -6834.144} C_VEL
LIN {X 0,Y 481.923,Z 226.941,A -85,B 0,C 180,E1 -6837.496,E2 -6837.496} C_VEL
LIN {X 0,Y 481.883,Z 226.949,A -85,B 0,C 180,E1 -6840.839,E2 -6840.839} C_VEL
LIN {X 0,Y 481.926,Z 226.949,A -85,B 0,C 180,E1 -6842.511,E2 -6842.511} C_VEL
LIN {X 0,Y 481.799,Z 226.972,A -85,B 0,C 180,E1 -6845.864,E2 -6845.864} C_VEL
LIN {X 0,Y 481.761,Z 226.963,A -85,B 0,C 180,E1 -6848.392,E2 -6848.392} C_VEL
LIN {X 0,Y 481.753,Z 226.963,A -85,B 0,C 180,E1 -6851.788,E2 -6851.788} C_VEL
LIN {X 0,Y 481.746,Z 226.971,A -85,B 0,C 180,E1 -6855.227,E2 -6855.227} C_VEL
LIN {X 0,Y 481.712,Z 226.974,A -85,B 0,C 180,E1 -6858.725,E2 -6858.725} C_VEL
LIN {X 0,Y 481.65,Z 226.974,A -85,B 0,C 180,E1 -6861.398,E2 -6861.398} C_VEL
LIN {X 0,Y 481.668,Z 226.982,A -85,B 0,C 180,E1 -6864.117,E2 -6864.117} C_VEL
LIN {X 0,Y 481.719,Z 226.977,A -85,B 0,C 180,E1 -6867.134,E2 -6867.134} C_VEL
LIN {X 0,Y 481.684,Z 226.971,A -85,B 0,C 180,E1 -6869.744,E2 -6869.744} C_VEL
LIN {X 0,Y 481.659,Z 226.986,A -85,B 0,C 180,E1 -6872.678,E2 -6872.678} C_VEL
LIN {X 0,Y 481.638,Z 226.984,A -85,B 0,C 180,E1 -6875.712,E2 -6875.712} C_VEL
LIN {X 0,Y 481.677,Z 226.982,A -85,B 0,C 180,E1 -6878.861,E2 -6878.861} C_VEL
LIN {X 0,Y 481.654,Z 226.981,A -85,B 0,C 180,E1 -6881.914,E2 -6881.914} C_VEL
LIN {X 0,Y 481.662,Z 226.969,A -85,B 0,C 180,E1 -6884.46,E2 -6884.46} C_VEL
LIN {X 0,Y 481.65,Z 226.988,A -85,B 0,C 180,E1 -6887.84,E2 -6887.84} C_VEL
LIN {X 0,Y 481.663,Z 226.981,A -85,B 0,C 180,E1 -6890.656,E2 -6890.656} C_VEL
LIN {X 0,Y 481.629,Z 226.988,A -85,B 0,C 180,E1 -6893.379,E2 -6893.379} C_VEL
LIN {X 0,Y 481.702,Z 226.981,A -85,B 0,C 180,E1 -6896.33,E2 -6896.33} C_VEL
LIN {X 0,Y 481.656,Z 226.985,A -85,B 0,C 180,E1 -6899.419,E2 -6899.419} C_VEL
LIN {X 0,Y 481.699,Z 226.985,A -85,B 0,C 180,E1 -6902.168,E2 -6902.168} C_VEL
LIN {X 0,Y 481.726,Z 227.083,A -85,B 0,C 180,E1 -6905.546,E2 -6905.546} C_VEL
LIN {X 0,Y 483.501,Z 237.281,A -85,B 0,C 180,E1 -6907.57,E2 -6907.57} C_VEL
LIN {X 0,Y 482.78,Z 256.879,A -85,B 0,C 180,E1 -6911.129,E2 -6911.129} C_VEL
LIN {X 0,Y 482.361,Z 270.336,A -85,B 0,C 180,E1 -6913.498,E2 -6913.498} C_VEL
LIN {X 0,Y 484.838,Z 286.524,A -85,B 0,C 180,E1 -6913.85,E2 -6913.85} C_VEL
LIN {X 0,Y 484.255,Z 377.914,A -85,B 0,C 180,E1 -6915.234,E2 -6915.234} C_VEL
LIN {X 0,Y 483.938,Z 391.213,A -85,B 0,C 180,E1 -6915.6,E2 -6915.6} C_VEL
LIN {X 0,Y 483.542,Z 403.964,A -85,B 0,C 180,E1 -6916.125,E2 -6916.125} C_VEL
LIN {X 0,Y 483.15,Z 415.608,A -85,B 0,C 180,E1 -6916.778,E2 -6916.778} C_VEL
LIN {X 0,Y 482.735,Z 426.969,A -85,B 0,C 180,E1 -6917.6,E2 -6917.6} C_VEL
LIN {X 0,Y 482.285,Z 437.458,A -85,B 0,C 180,E1 -6918.548,E2 -6918.548} C_VEL
LIN {X 0,Y 481.879,Z 446.029,A -85,B 0,C 180,E1 -6919.496,E2 -6919.496} C_VEL
LIN {X 0,Y 481.534,Z 453.932,A -85,B 0,C 180,E1 -6920.55,E2 -6920.55} C_VEL
LIN {X 0,Y 481.259,Z 461.651,A -85,B 0,C 180,E1 -6921.815,E2 -6921.815} C_VEL
LIN {X 0,Y 481.02,Z 468.753,A -85,B 0,C 180,E1 -6923.288,E2 -6923.288} C_VEL
LIN {X 0,Y 480.963,Z 473.479,A -85,B 0,C 180,E1 -6924.55,E2 -6924.55} C_VEL
LIN {X 0,Y 480.83,Z 477.088,A -85,B 0,C 180,E1 -6925.809,E2 -6925.809} C_VEL
LIN {X 0,Y 480.873,Z 478.952,A -85,B 0,C 180,E1 -6926.649,E2 -6926.649} C_VEL
LIN {X 0,Y 480.792,Z 481.343,A -85,B 0,C 180,E1 -6928.325,E2 -6928.325} C_VEL
LIN {X 0,Y 480.745,Z 482.169,A -85,B 0,C 180,E1 -6930,E2 -6930} C_VEL
LIN {X 0,Y 480.762,Z 481.955,A -85,B 0,C 180,E1 -6930.838,E2 -6930.838} C_VEL
LIN {X 0,Y 480.792,Z 481.35,A -85,B 0,C 180,E1 -6931.676,E2 -6931.676} C_VEL
LIN {X 0,Y 480.873,Z 478.966,A -85,B 0,C 180,E1 -6933.352,E2 -6933.352} C_VEL
LIN {X 0,Y 480.842,Z 476.037,A -85,B 0,C 180,E1 -6934.611,E2 -6934.611} C_VEL
LIN {X 0,Y 480.964,Z 472.073,A -85,B 0,C 180,E1 -6935.871,E2 -6935.871} C_VEL
LIN {X 0,Y 481.114,Z 465.976,A -85,B 0,C 180,E1 -6937.344,E2 -6937.344} C_VEL
LIN {X 0,Y 481.36,Z 459.312,A -85,B 0,C 180,E1 -6938.607,E2 -6938.607} C_VEL
LIN {X 0,Y 481.695,Z 451.042,A -85,B 0,C 180,E1 -6939.871,E2 -6939.871} C_VEL
LIN {X 0,Y 482.023,Z 442.577,A -85,B 0,C 180,E1 -6940.926,E2 -6940.926} C_VEL
LIN {X 0,Y 482.568,Z 432.123,A -85,B 0,C 180,E1 -6941.978,E2 -6941.978} C_VEL
LIN {X 0,Y 482.908,Z 420.732,A -85,B 0,C 180,E1 -6942.902,E2 -6942.902} C_VEL
LIN {X 0,Y 483.399,Z 408.554,A -85,B 0,C 180,E1 -6943.666,E2 -6943.666} C_VEL
LIN {X 0,Y 483.807,Z 396.284,A -85,B 0,C 180,E1 -6944.244,E2 -6944.244} C_VEL
LIN {X 0,Y 484.202,Z 382.773,A -85,B 0,C 180,E1 -6944.688,E2 -6944.688} C_VEL
LIN {X 0,Y 484.435,Z 367.319,A -85,B 0,C 180,E1 -6944.976,E2 -6944.976} C_VEL
LIN {X 0,Y 484.921,Z 285.518,A -85,B 0,C 180,E1 -6946.205,E2 -6946.205} C_VEL
LIN {X 0,Y 482.389,Z 270.526,A -85,B 0,C 180,E1 -6946.543,E2 -6946.543} C_VEL
LIN {X 0,Y 482.365,Z 269.048,A -85,B 0,C 180,E1 -6946.724,E2 -6946.724} C_VEL
LIN {X 0,Y 482.898,Z 253.294,A -85,B 0,C 180,E1 -6949.557,E2 -6949.557} C_VEL
LIN {X 0,Y 483.567,Z 237.541,A -85,B 0,C 180,E1 -6952.427,E2 -6952.427} C_VEL
LIN {X 0,Y 481.754,Z 227.325,A -85,B 0,C 180,E1 -6954.453,E2 -6954.453} C_VEL
LIN {X 0,Y 481.689,Z 227.019,A -85,B 0,C 180,E1 -6954.571,E2 -6954.571} C_VEL
LIN {X 0,Y 481.701,Z 226.984,A -85,B 0,C 180,E1 -6957.832,E2 -6957.832} C_VEL
LIN {X 0,Y 481.653,Z 226.984,A -85,B 0,C 180,E1 -6960.711,E2 -6960.711} C_VEL
LIN {X 0,Y 481.709,Z 226.979,A -85,B 0,C 180,E1 -6963.732,E2 -6963.732} C_VEL
LIN {X 0,Y 481.63,Z 226.989,A -85,B 0,C 180,E1 -6966.747,E2 -6966.747} C_VEL
LIN {X 0,Y 481.668,Z 226.984,A -85,B 0,C 180,E1 -6969.941,E2 -6969.941} C_VEL
LIN {X 0,Y 481.637,Z 226.983,A -85,B 0,C 180,E1 -6973.145,E2 -6973.145} C_VEL
LIN {X 0,Y 481.664,Z 226.983,A -85,B 0,C 180,E1 -6975.64,E2 -6975.64} C_VEL
LIN {X 0,Y 481.658,Z 226.987,A -85,B 0,C 180,E1 -6978.956,E2 -6978.956} C_VEL
LIN {X 0,Y 481.659,Z 226.982,A -85,B 0,C 180,E1 -6981.992,E2 -6981.992} C_VEL
LIN {X 0,Y 481.691,Z 226.981,A -85,B 0,C 180,E1 -6985.315,E2 -6985.315} C_VEL
LIN {X 0,Y 481.652,Z 226.982,A -85,B 0,C 180,E1 -6988.309,E2 -6988.309} C_VEL
LIN {X 0,Y 481.669,Z 226.984,A -85,B 0,C 180,E1 -6991.214,E2 -6991.214} C_VEL
LIN {X 0,Y 481.652,Z 226.984,A -85,B 0,C 180,E1 -6994.037,E2 -6994.037} C_VEL
LIN {X 0,Y 481.662,Z 226.983,A -85,B 0,C 180,E1 -6996.815,E2 -6996.815} C_VEL
LIN {X 0,Y 481.704,Z 226.979,A -85,B 0,C 180,E1 -6999.5,E2 -6999.5} C_VEL
LIN {X 0,Y 481.699,Z 226.978,A -85,B 0,C 180,E1 -7002.155,E2 -7002.155} C_VEL
LIN {X 0,Y 481.749,Z 226.967,A -85,B 0,C 180,E1 -7004.773,E2 -7004.773} C_VEL
LIN {X 0,Y 481.757,Z 226.969,A -85,B 0,C 180,E1 -7008.212,E2 -7008.212} C_VEL
LIN {X 0,Y 481.734,Z 226.98,A -85,B 0,C 180,E1 -7011.608,E2 -7011.608} C_VEL
LIN {X 0,Y 481.8,Z 226.968,A -85,B 0,C 180,E1 -7014.136,E2 -7014.136} C_VEL
LIN {X 0,Y 481.918,Z 226.953,A -85,B 0,C 180,E1 -7017.489,E2 -7017.489} C_VEL
LIN {X 0,Y 481.94,Z 226.953,A -85,B 0,C 180,E1 -7019.996,E2 -7019.996} C_VEL
LIN {X 0,Y 481.918,Z 226.95,A -85,B 0,C 180,E1 -7022.504,E2 -7022.504} C_VEL
LIN {X 0,Y 481.794,Z 226.969,A -85,B 0,C 180,E1 -7025.857,E2 -7025.857} C_VEL
LIN {X 0,Y 481.736,Z 226.979,A -85,B 0,C 180,E1 -7028.385,E2 -7028.385} C_VEL
LIN {X 0,Y 481.744,Z 226.969,A -85,B 0,C 180,E1 -7031.781,E2 -7031.781} C_VEL
LIN {X 0,Y 481.735,Z 226.972,A -85,B 0,C 180,E1 -7035.22,E2 -7035.22} C_VEL
LIN {X 0,Y 481.697,Z 226.983,A -85,B 0,C 180,E1 -7038.717,E2 -7038.717} C_VEL
LIN {X 0,Y 481.636,Z 226.985,A -85,B 0,C 180,E1 -7041.39,E2 -7041.39} C_VEL
LIN {X 0,Y 481.662,Z 226.983,A -85,B 0,C 180,E1 -7044.109,E2 -7044.109} C_VEL
LIN {X 0,Y 481.729,Z 226.975,A -85,B 0,C 180,E1 -7047.135,E2 -7047.135} C_VEL
LIN {X 0,Y 481.658,Z 226.982,A -85,B 0,C 180,E1 -7049.737,E2 -7049.737} C_VEL
LIN {X 0,Y 481.65,Z 226.985,A -85,B 0,C 180,E1 -7052.67,E2 -7052.67} C_VEL
LIN {X 0,Y 481.617,Z 226.993,A -85,B 0,C 180,E1 -7055.705,E2 -7055.705} C_VEL
LIN {X 0,Y 481.695,Z 226.984,A -85,B 0,C 180,E1 -7059.351,E2 -7059.351} C_VEL
LIN {X 0,Y 481.645,Z 226.988,A -85,B 0,C 180,E1 -7062.153,E2 -7062.153} C_VEL
LIN {X 0,Y 481.628,Z 226.989,A -85,B 0,C 180,E1 -7064.453,E2 -7064.453} C_VEL
LIN {X 0,Y 481.655,Z 226.987,A -85,B 0,C 180,E1 -7066.842,E2 -7066.842} C_VEL
LIN {X 0,Y 481.708,Z 227.118,A -85,B 0,C 180,E1 -7069.603,E2 -7069.603} C_VEL
LIN {X 0,Y 482.871,Z 233.34,A -85,B 0,C 180,E1 -7070.904,E2 -7070.904} C_VEL
LIN {X 0,Y 482.874,Z 240.699,A -85,B 0,C 180,E1 -7072.317,E2 -7072.317} C_VEL
LIN {X 0,Y 482.413,Z 255.661,A -85,B 0,C 180,E1 -7075.14,E2 -7075.14} C_VEL
LIN {X 0,Y 482.412,Z 257.882,A -85,B 0,C 180,E1 -7075.493,E2 -7075.493} C_VEL
LIN {X 0,Y 485.002,Z 272.46,A -85,B 0,C 180,E1 -7075.837,E2 -7075.837} C_VEL
LIN {X 0,Y 484.434,Z 349.085,A -85,B 0,C 180,E1 -7076.986,E2 -7076.986} C_VEL
LIN {X 0,Y 483.74,Z 354.925,A -85,B 0,C 180,E1 -7077.049,E2 -7077.049} C_VEL
LIN {X 0,Y 480.87,Z 364.402,A -85,B 0,C 180,E1 -7077.115,E2 -7077.115} C_VEL
LIN {X 0,Y 477.944,Z 373.783,A -85,B 0,C 180,E1 -7077.261,E2 -7077.261} C_VEL
LIN {X 0,Y 477.152,Z 379.469,A -85,B 0,C 180,E1 -7077.429,E2 -7077.429} C_VEL
LIN {X 0,Y 476.789,Z 391.605,A -85,B 0,C 180,E1 -7077.951,E2 -7077.951} C_VEL
LIN {X 0,Y 476.432,Z 402.202,A -85,B 0,C 180,E1 -7078.558,E2 -7078.558} C_VEL
LIN {X 0,Y 475.956,Z 413.383,A -85,B 0,C 180,E1 -7079.374,E2 -7079.374} C_VEL
LIN {X 0,Y 475.467,Z 423.756,A -85,B 0,C 180,E1 -7080.319,E2 -7080.319} C_VEL
LIN {X 0,Y 475.093,Z 432.245,A -85,B 0,C 180,E1 -7081.264,E2 -7081.264} C_VEL
LIN {X 0,Y 474.656,Z 440.953,A -85,B 0,C 180,E1 -7082.438,E2 -7082.438} C_VEL
LIN {X 0,Y 474.282,Z 448.006,A -85,B 0,C 180,E1 -7083.606,E2 -7083.606} C_VEL
LIN {X 0,Y 474.065,Z 455.118,A -85,B 0,C 180,E1 -7085.091,E2 -7085.091} C_VEL
LIN {X 0,Y 473.89,Z 459.994,A -85,B 0,C 180,E1 -7086.395,E2 -7086.395} C_VEL
LIN {X 0,Y 473.776,Z 463.91,A -85,B 0,C 180,E1 -7087.773,E2 -7087.773} C_VEL
LIN {X 0,Y 473.679,Z 466.687,A -85,B 0,C 180,E1 -7089.167,E2 -7089.167} C_VEL
LIN {X 0,Y 473.659,Z 467.868,A -85,B 0,C 180,E1 -7090.046,E2 -7090.046} C_VEL
LIN {X 0,Y 473.62,Z 468.899,A -85,B 0,C 180,E1 -7091.728,E2 -7091.728} C_VEL
LIN {X 0,Y 473.617,Z 468.813,A -85,B 0,C 180,E1 -7092.736,E2 -7092.736} C_VEL
LIN {X 0,Y 473.62,Z 468.231,A -85,B 0,C 180,E1 -7093.624,E2 -7093.624} C_VEL
LIN {X 0,Y 473.688,Z 467.064,A -85,B 0,C 180,E1 -7094.639,E2 -7094.639} C_VEL
LIN {X 0,Y 473.724,Z 465.828,A -85,B 0,C 180,E1 -7095.392,E2 -7095.392} C_VEL
LIN {X 0,Y 473.805,Z 462.845,A -85,B 0,C 180,E1 -7096.708,E2 -7096.708} C_VEL
LIN {X 0,Y 473.935,Z 458.396,A -85,B 0,C 180,E1 -7098.126,E2 -7098.126} C_VEL
LIN {X 0,Y 474.151,Z 452.539,A -85,B 0,C 180,E1 -7099.538,E2 -7099.538} C_VEL
LIN {X 0,Y 474.419,Z 445.731,A -85,B 0,C 180,E1 -7100.836,E2 -7100.836} C_VEL
LIN {X 0,Y 474.78,Z 437.284,A -85,B 0,C 180,E1 -7102.13,E2 -7102.13} C_VEL
LIN {X 0,Y 475.127,Z 428.598,A -85,B 0,C 180,E1 -7103.204,E2 -7103.204} C_VEL
LIN {X 0,Y 475.6,Z 417.906,A -85,B 0,C 180,E1 -7104.275,E2 -7104.275} C_VEL
LIN {X 0,Y 476.126,Z 407.246,A -85,B 0,C 180,E1 -7105.131,E2 -7105.131} C_VEL
LIN {X 0,Y 476.589,Z 395.364,A -85,B 0,C 180,E1 -7105.877,E2 -7105.877} C_VEL
LIN {X 0,Y 476.958,Z 383.036,A -85,B 0,C 180,E1 -7106.462,E2 -7106.462} C_VEL
LIN {X 0,Y 477.223,Z 370.39,A -85,B 0,C 180,E1 -7106.887,E2 -7106.887} C_VEL
LIN {X 0,Y 477.419,Z 355.382,A -85,B 0,C 180,E1 -7107.178,E2 -7107.178} C_VEL
LIN {X 0,Y 477.929,Z 272.505,A -85,B 0,C 180,E1 -7108.433,E2 -7108.433} C_VEL
LIN {X 0,Y 475.362,Z 258.097,A -85,B 0,C 180,E1 -7108.768,E2 -7108.768} C_VEL
LIN {X 0,Y 475.642,Z 249.348,A -85,B 0,C 180,E1 -7110.423,E2 -7110.423} C_VEL
LIN {X 0,Y 476.152,Z 236.518,A -85,B 0,C 180,E1 -7112.961,E2 -7112.961} C_VEL
LIN {X 0,Y 474.74,Z 227.937,A -85,B 0,C 180,E1 -7114.803,E2 -7114.803} C_VEL
LIN {X 0,Y 474.754,Z 227.845,A -85,B 0,C 180,E1 -7117.656,E2 -7117.656} C_VEL
LIN {X 0,Y 474.676,Z 227.856,A -85,B 0,C 180,E1 -7121.097,E2 -7121.097} C_VEL
LIN {X 0,Y 474.654,Z 227.856,A -85,B 0,C 180,E1 -7123.704,E2 -7123.704} C_VEL
LIN {X 0,Y 474.615,Z 227.863,A -85,B 0,C 180,E1 -7126.34,E2 -7126.34} C_VEL
LIN {X 0,Y 474.623,Z 227.855,A -85,B 0,C 180,E1 -7129.012,E2 -7129.012} C_VEL
LIN {X 0,Y 474.63,Z 227.858,A -85,B 0,C 180,E1 -7131.726,E2 -7131.726} C_VEL
LIN {X 0,Y 474.633,Z 227.857,A -85,B 0,C 180,E1 -7134.494,E2 -7134.494} C_VEL
LIN {X 0,Y 474.653,Z 227.846,A -85,B 0,C 180,E1 -7137.341,E2 -7137.341} C_VEL
LIN {X 0,Y 474.604,Z 227.863,A -85,B 0,C 180,E1 -7140.822,E2 -7140.822} C_VEL
LIN {X 0,Y 474.611,Z 227.868,A -85,B 0,C 180,E1 -7143.222,E2 -7143.222} C_VEL
LIN {X 0,Y 474.569,Z 227.864,A -85,B 0,C 180,E1 -7146.325,E2 -7146.325} C_VEL
LIN {X 0,Y 474.65,Z 227.863,A -85,B 0,C 180,E1 -7149.545,E2 -7149.545} C_VEL
LIN {X 0,Y 474.65,Z 227.847,A -85,B 0,C 180,E1 -7152.93,E2 -7152.93} C_VEL
LIN {X 0,Y 474.664,Z 227.856,A -85,B 0,C 180,E1 -7156.51,E2 -7156.51} C_VEL
LIN {X 0,Y 474.609,Z 227.858,A -85,B 0,C 180,E1 -7159.349,E2 -7159.349} C_VEL
LIN {X 0,Y 474.591,Z 227.854,A -85,B 0,C 180,E1 -7161.706,E2 -7161.706} C_VEL
LIN {X 0,Y 474.606,Z 227.863,A -85,B 0,C 180,E1 -7164.731,E2 -7164.731} C_VEL
LIN {X 0,Y 474.613,Z 227.861,A -85,B 0,C 180,E1 -7167.792,E2 -7167.792} C_VEL
LIN {X 0,Y 474.609,Z 227.852,A -85,B 0,C 180,E1 -7170.887,E2 -7170.887} C_VEL
LIN {X 0,Y 474.645,Z 227.845,A -85,B 0,C 180,E1 -7173.633,E2 -7173.633} C_VEL
LIN {X 0,Y 474.617,Z 227.864,A -85,B 0,C 180,E1 -7176.645,E2 -7176.645} C_VEL
LIN {X 0,Y 474.659,Z 227.857,A -85,B 0,C 180,E1 -7179.19,E2 -7179.19} C_VEL
LIN {X 0,Y 474.643,Z 227.85,A -85,B 0,C 180,E1 -7181.889,E2 -7181.889} C_VEL
LIN {X 0,Y 474.687,Z 227.838,A -85,B 0,C 180,E1 -7184.549,E2 -7184.549} C_VEL
LIN {X 0,Y 474.729,Z 227.841,A -85,B 0,C 180,E1 -7188.043,E2 -7188.043} C_VEL
LIN {X 0,Y 474.721,Z 227.853,A -85,B 0,C 180,E1 -7191.491,E2 -7191.491} C_VEL
LIN {X 0,Y 474.775,Z 227.836,A -85,B 0,C 180,E1 -7194.056,E2 -7194.056} C_VEL
LIN {X 0,Y 474.889,Z 227.816,A -85,B 0,C 180,E1 -7197.459,E2 -7197.459} C_VEL
LIN {X 0,Y 474.908,Z 227.822,A -85,B 0,C 180,E1 -7200.004,E2 -7200.004} C_VEL
LIN {X 0,Y 474.892,Z 227.825,A -85,B 0,C 180,E1 -7202.548,E2 -7202.548} C_VEL
LIN {X 0,Y 474.76,Z 227.847,A -85,B 0,C 180,E1 -7205.951,E2 -7205.951} C_VEL
LIN {X 0,Y 474.727,Z 227.837,A -85,B 0,C 180,E1 -7208.517,E2 -7208.517} C_VEL
LIN {X 0,Y 474.706,Z 227.843,A -85,B 0,C 180,E1 -7211.966,E2 -7211.966} C_VEL
LIN {X 0,Y 474.703,Z 227.849,A -85,B 0,C 180,E1 -7215.459,E2 -7215.459} C_VEL
LIN {X 0,Y 474.667,Z 227.848,A -85,B 0,C 180,E1 -7219.013,E2 -7219.013} C_VEL
LIN {X 0,Y 474.593,Z 227.853,A -85,B 0,C 180,E1 -7221.732,E2 -7221.732} C_VEL
LIN {X 0,Y 474.645,Z 227.861,A -85,B 0,C 180,E1 -7224.497,E2 -7224.497} C_VEL
LIN {X 0,Y 474.68,Z 227.852,A -85,B 0,C 180,E1 -7227.335,E2 -7227.335} C_VEL
LIN {X 0,Y 474.61,Z 227.853,A -85,B 0,C 180,E1 -7230.233,E2 -7230.233} C_VEL
LIN {X 0,Y 474.621,Z 227.866,A -85,B 0,C 180,E1 -7233.225,E2 -7233.225} C_VEL
LIN {X 0,Y 474.591,Z 227.861,A -85,B 0,C 180,E1 -7236.326,E2 -7236.326} C_VEL
LIN {X 0,Y 474.633,Z 227.863,A -85,B 0,C 180,E1 -7239.55,E2 -7239.55} C_VEL
LIN {X 0,Y 474.608,Z 227.857,A -85,B 0,C 180,E1 -7242.235,E2 -7242.235} C_VEL
LIN {X 0,Y 474.624,Z 227.848,A -85,B 0,C 180,E1 -7245.3,E2 -7245.3} C_VEL
LIN {X 0,Y 474.623,Z 227.86,A -85,B 0,C 180,E1 -7248.215,E2 -7248.215} C_VEL
LIN {X 0,Y 474.616,Z 227.863,A -85,B 0,C 180,E1 -7251.544,E2 -7251.544} C_VEL
LIN {X 0,Y 474.63,Z 227.858,A -85,B 0,C 180,E1 -7254.727,E2 -7254.727} C_VEL
LIN {X 0,Y 474.643,Z 227.864,A -85,B 0,C 180,E1 -7257.789,E2 -7257.789} C_VEL
LIN {X 0,Y 474.629,Z 227.861,A -85,B 0,C 180,E1 -7260.887,E2 -7260.887} C_VEL
LIN {X 0,Y 474.635,Z 227.864,A -85,B 0,C 180,E1 -7263.627,E2 -7263.627} C_VEL
LIN {X 0,Y 474.674,Z 228.009,A -85,B 0,C 180,E1 -7265.392,E2 -7265.392} C_VEL
LIN {X 0,Y 476.527,Z 238.294,A -85,B 0,C 180,E1 -7267.452,E2 -7267.452} C_VEL
LIN {X 0,Y 475.856,Z 255.576,A -85,B 0,C 180,E1 -7270.636,E2 -7270.636} C_VEL
LIN {X 0,Y 475.35,Z 270.229,A -85,B 0,C 180,E1 -7273.26,E2 -7273.26} C_VEL
LIN {X 0,Y 477.848,Z 285.742,A -85,B 0,C 180,E1 -7273.612,E2 -7273.612} C_VEL
LIN {X 0,Y 477.521,Z 363.942,A -85,B 0,C 180,E1 -7274.802,E2 -7274.802} C_VEL
LIN {X 0,Y 477.294,Z 381.81,A -85,B 0,C 180,E1 -7275.122,E2 -7275.122} C_VEL
LIN {X 0,Y 476.983,Z 393.776,A -85,B 0,C 180,E1 -7275.494,E2 -7275.494} C_VEL
LIN {X 0,Y 476.556,Z 405.697,A -85,B 0,C 180,E1 -7276.026,E2 -7276.026} C_VEL
LIN {X 0,Y 476.169,Z 416.586,A -85,B 0,C 180,E1 -7276.667,E2 -7276.667} C_VEL
LIN {X 0,Y 475.717,Z 428.159,A -85,B 0,C 180,E1 -7277.535,E2 -7277.535} C_VEL
LIN {X 0,Y 475.244,Z 438.305,A -85,B 0,C 180,E1 -7278.484,E2 -7278.484} C_VEL
LIN {X 0,Y 474.795,Z 447.544,A -85,B 0,C 180,E1 -7279.553,E2 -7279.553} C_VEL
LIN {X 0,Y 474.391,Z 456.524,A -85,B 0,C 180,E1 -7280.836,E2 -7280.836} C_VEL
LIN {X 0,Y 474.112,Z 463.753,A -85,B 0,C 180,E1 -7282.119,E2 -7282.119} C_VEL
LIN {X 0,Y 473.906,Z 470.002,A -85,B 0,C 180,E1 -7283.527,E2 -7283.527} C_VEL
LIN {X 0,Y 473.839,Z 474.681,A -85,B 0,C 180,E1 -7284.895,E2 -7284.895} C_VEL
LIN {X 0,Y 473.737,Z 476.979,A -85,B 0,C 180,E1 -7285.746,E2 -7285.746} C_VEL
LIN {X 0,Y 473.768,Z 478.845,A -85,B 0,C 180,E1 -7286.599,E2 -7286.599} C_VEL
LIN {X 0,Y 473.725,Z 480.244,A -85,B 0,C 180,E1 -7287.449,E2 -7287.449} C_VEL
LIN {X 0,Y 473.69,Z 481.851,A -85,B 0,C 180,E1 -7289.15,E2 -7289.15} C_VEL
LIN {X 0,Y 473.672,Z 482.071,A -85,B 0,C 180,E1 -7290,E2 -7290} C_VEL
LIN {X 0,Y 473.69,Z 481.859,A -85,B 0,C 180,E1 -7290.85,E2 -7290.85} C_VEL
LIN {X 0,Y 473.725,Z 480.263,A -85,B 0,C 180,E1 -7292.551,E2 -7292.551} C_VEL
LIN {X 0,Y 473.768,Z 478.875,A -85,B 0,C 180,E1 -7293.402,E2 -7293.402} C_VEL
LIN {X 0,Y 473.766,Z 475.95,A -85,B 0,C 180,E1 -7294.68,E2 -7294.68} C_VEL
LIN {X 0,Y 473.868,Z 471.993,A -85,B 0,C 180,E1 -7295.959,E2 -7295.959} C_VEL
LIN {X 0,Y 474.036,Z 465.911,A -85,B 0,C 180,E1 -7297.454,E2 -7297.454} C_VEL
LIN {X 0,Y 474.325,Z 459.263,A -85,B 0,C 180,E1 -7298.736,E2 -7298.736} C_VEL
LIN {X 0,Y 474.678,Z 451.015,A -85,B 0,C 180,E1 -7300.019,E2 -7300.019} C_VEL
LIN {X 0,Y 475.052,Z 442.57,A -85,B 0,C 180,E1 -7301.089,E2 -7301.089} C_VEL
LIN {X 0,Y 475.609,Z 432.288,A -85,B 0,C 180,E1 -7302.142,E2 -7302.142} C_VEL
LIN {X 0,Y 475.996,Z 420.55,A -85,B 0,C 180,E1 -7303.11,E2 -7303.11} C_VEL
LIN {X 0,Y 476.522,Z 408.652,A -85,B 0,C 180,E1 -7303.867,E2 -7303.867} C_VEL
LIN {X 0,Y 476.951,Z 396.443,A -85,B 0,C 180,E1 -7304.453,E2 -7304.453} C_VEL
LIN {X 0,Y 477.367,Z 383.08,A -85,B 0,C 180,E1 -7304.903,E2 -7304.903} C_VEL
LIN {X 0,Y 477.599,Z 367.938,A -85,B 0,C 180,E1 -7305.196,E2 -7305.196} C_VEL
LIN {X 0,Y 478.138,Z 286.315,A -85,B 0,C 180,E1 -7306.442,E2 -7306.442} C_VEL
LIN {X 0,Y 475.431,Z 270.361,A -85,B 0,C 180,E1 -7306.809,E2 -7306.809} C_VEL
LIN {X 0,Y 475.418,Z 267.836,A -85,B 0,C 180,E1 -7307.197,E2 -7307.197} C_VEL
LIN {X 0,Y 476.045,Z 252.082,A -85,B 0,C 180,E1 -7310.075,E2 -7310.075} C_VEL
LIN {X 0,Y 476.626,Z 238.76,A -85,B 0,C 180,E1 -7312.543,E2 -7312.543} C_VEL
LIN {X 0,Y 474.894,Z 229.121,A -85,B 0,C 180,E1 -7314.48,E2 -7314.48} C_VEL
LIN {X 0,Y 474.654,Z 227.888,A -85,B 0,C 180,E1 -7314.814,E2 -7314.814} C_VEL
LIN {X 0,Y 474.685,Z 227.858,A -85,B 0,C 180,E1 -7317.332,E2 -7317.332} C_VEL
LIN {X 0,Y 474.613,Z 227.864,A -85,B 0,C 180,E1 -7320.23,E2 -7320.23} C_VEL
LIN {X 0,Y 474.645,Z 227.855,A -85,B 0,C 180,E1 -7323.22,E2 -7323.22} C_VEL
LIN {X 0,Y 474.594,Z 227.869,A -85,B 0,C 180,E1 -7326.323,E2 -7326.323} C_VEL
LIN {X 0,Y 474.632,Z 227.856,A -85,B 0,C 180,E1 -7329.547,E2 -7329.547} C_VEL
LIN {X 0,Y 474.608,Z 227.862,A -85,B 0,C 180,E1 -7332.232,E2 -7332.232} C_VEL
LIN {X 0,Y 474.627,Z 227.859,A -85,B 0,C 180,E1 -7335.297,E2 -7335.297} C_VEL
LIN {X 0,Y 474.625,Z 227.854,A -85,B 0,C 180,E1 -7338.212,E2 -7338.212} C_VEL
LIN {X 0,Y 474.619,Z 227.858,A -85,B 0,C 180,E1 -7341.541,E2 -7341.541} C_VEL
LIN {X 0,Y 474.629,Z 227.863,A -85,B 0,C 180,E1 -7344.723,E2 -7344.723} C_VEL
